(* ADS write *)
_fbWriteProp(
	BACnetDevicePort	:= stAdsConn.nAmsPort,
	bExecute			:= ,
	sNetId				:= stAdsConn.sAmsNetId,
	ObjectType			:= F_BACnet_GetObjType(tObjectID),
	PropertyID			:= BACnetPropertyIdentifier_RecipientList,
	Priority			:= BACnetPriority_None,
	DataType			:= BACnetDataType_RecipientArr,
	ObjectInstance		:= F_BACnet_GetObjInstance(tObjectID),
	ptrValue			:= ADR(stBACnet_AdsBuffer.arrData),
	nLenValue			:= TO_UDINT(_iDataEntry) * TO_UDINT(_cbDestListElem),
	bDone				=> ,
	bBusy				=> ,
	bError				=> ,
	nErrID				=> );

(* trigger start event *)
_rtrigGet(CLK:= bGet, Q=> );
_rtrigSet(CLK:= bSet, Q=> );

(* state machine *)
CASE _i OF

	0: (* Idle *)
		IF 		_rtrigGet.Q
			OR	_rtrigSet.Q
			OR	(		(		(_nAdsReloadOld <> stAdsConn.nReload)
							OR	(_tObjectIDOld <> tObjectID)
						)
					AND	bAutoGet
				)
		THEN
			IF (NOT stAdsConn.bValid) THEN
				(* ADS connection not valid *)
				nErrorId := BACnet_ERR_INVALID_ADS_CONN;
			ELSIF (NOT stAdsConn.bServer AND NOT stAdsConn.bClient) THEN
				(* not a server nor a client *)
				nErrorId := BACnet_ERR_ADS_NoServerClient;
			ELSE
				(* decide get or set *)
				IF _rtrigGet.Q THEN
					_i := 1;
				ELSIF _rtrigSet.Q THEN
					_i := 11;
				ELSIF bAutoGet THEN
					_i := 1;
				END_IF
				nErrorId := BACnet_ERR_NO_ERROR;
				(* reset index *)
				_iEntry	:= 0;
				(* initialize pointer *)
				_pEntryList := ADR(stBACnet_AdsBuffer.arrData);
				(* remind parameter *)
				_tObjectIDOld := tObjectID;
				_nAdsReloadOld := stAdsConn.nReload;
			END_IF
			(* reset done flag *)
			bDone := FALSE;
		END_IF
		IF (NOT bGet) AND (NOT bSet) AND (NOT bAutoGet) THEN
			nErrorId := BACnet_ERR_NO_ERROR;
			bDone := FALSE;
		END_IF

	(* READ *)
	1: (* read object property data via ADS *)
		IF TestAndSet(stBACnet_AdsBuffer.bTestSet) THEN
			IF _fbReadProp.bExecute THEN
				IF _fbReadProp.bError THEN
					_i := 100;
					nErrorId := BACnet_ERR_ADS_Read;
					_fbReadProp.bExecute := FALSE;
				ELSIF (NOT _fbReadProp.bBusy) THEN
					_i := 2;
					_fbReadProp.bExecute := FALSE;
					(* clear output data *)
					MEMSET(ADR(stRecipients), 0, SIZEOF(stRecipients));
					(* check array size *)
					_cbDestList 	:= SIZEOF(_pEntryList^);
					_cbDestListElem	:= SIZEOF(_pEntryList^[0]);
					_iEntryCheck := MIN(_fbReadProp.nProcessedLen, _cbDestList) MOD _cbDestListElem;
					IF (_iEntryCheck <> 0) OR (_cbDestListElem = 0) THEN
						_i := 100;
						nErrorId := BACnet_ERR_ADS_WrongEntrySize;
					ELSE
						(* scan property *)
						_iDataEntry := 0;
						_iReadElems := MIN(32767, MIN(_fbReadProp.nProcessedLen, _cbDestList) / _cbDestListElem);
						FOR _iEntry := 0 TO UDINT_TO_INT(_iReadElems) - 1 DO
							IF		(_pEntryList^[_iEntry].stRecipient.eRecipientChoice = BACnetRecipientChoice_device)
								AND	(F_BACnet_GetObjType(_pEntryList^[_iEntry].stRecipient.tDeviceId) = BACnetObjectType_Device)
							THEN
								stRecipients.arrDestList[_iDataEntry].stFromTime	:= _pEntryList^[_iEntry].stFromTime;
								stRecipients.arrDestList[_iDataEntry].stToTime	:= _pEntryList^[_iEntry].stToTime;
								stRecipients.arrDestList[_iDataEntry].tDeviceId	:= _pEntryList^[_iEntry].stRecipient.tDeviceId;
								stRecipients.arrDestList[_iDataEntry].nProcessId	:= _pEntryList^[_iEntry].nProcessId;
								stRecipients.arrDestList[_iDataEntry].bMonday		:= _F_BACnet_IsBitFieldBitSet(_pEntryList^[_iEntry].nValidDaysFlags, BACnetDaysOfWeekBits_Monday);
								stRecipients.arrDestList[_iDataEntry].bTuesday	:= _F_BACnet_IsBitFieldBitSet(_pEntryList^[_iEntry].nValidDaysFlags, BACnetDaysOfWeekBits_Tuesday);
								stRecipients.arrDestList[_iDataEntry].bWednesday	:= _F_BACnet_IsBitFieldBitSet(_pEntryList^[_iEntry].nValidDaysFlags, BACnetDaysOfWeekBits_Wednesday);
								stRecipients.arrDestList[_iDataEntry].bThursday	:= _F_BACnet_IsBitFieldBitSet(_pEntryList^[_iEntry].nValidDaysFlags, BACnetDaysOfWeekBits_Thursday);
								stRecipients.arrDestList[_iDataEntry].bFriday		:= _F_BACnet_IsBitFieldBitSet(_pEntryList^[_iEntry].nValidDaysFlags, BACnetDaysOfWeekBits_Friday);
								stRecipients.arrDestList[_iDataEntry].bSaturday	:= _F_BACnet_IsBitFieldBitSet(_pEntryList^[_iEntry].nValidDaysFlags, BACnetDaysOfWeekBits_Saturday);
								stRecipients.arrDestList[_iDataEntry].bSunday		:= _F_BACnet_IsBitFieldBitSet(_pEntryList^[_iEntry].nValidDaysFlags, BACnetDaysOfWeekBits_Sunday);
								stRecipients.arrDestList[_iDataEntry].bToNormal	:= _F_BACnet_IsBitFieldBitSet(_pEntryList^[_iEntry].nEventTransBits, BACnetEventTransitionBit_to_normal);
								stRecipients.arrDestList[_iDataEntry].bToOffNormal:= _F_BACnet_IsBitFieldBitSet(_pEntryList^[_iEntry].nEventTransBits, BACnetEventTransitionBit_to_offnormal);
								stRecipients.arrDestList[_iDataEntry].bToFault	:= _F_BACnet_IsBitFieldBitSet(_pEntryList^[_iEntry].nEventTransBits, BACnetEventTransitionBit_to_fault);
								stRecipients.arrDestList[_iDataEntry].bIssueConfirmedNotification	:= _pEntryList^[_iEntry].bIssueConfNot;
								_iDataEntry := _iDataEntry + 1;
							END_IF
						END_FOR
						(* calculate entry count *)
						stRecipients.nEntries := _iDataEntry;
						_i := 100;
					END_IF
				END_IF

			ELSIF (stBACnet_AdsBuffer.iLocked = 0) THEN
				_fbReadProp.bExecute := TRUE;
				(* lock global ADS buffer *)
				stBACnet_AdsBuffer.iLocked := SIZEOF(stBACnet_AdsBuffer.arrData);
			END_IF

			(* release temporary task lock *)
			stBACnet_AdsBuffer.bTestSet := FALSE;
		END_IF


	(* WRITE *)
	11: (* lock global ADS buffer *)
		IF TestAndSet(stBACnet_AdsBuffer.bTestSet) THEN
			IF stBACnet_AdsBuffer.iLocked = 0 THEN
				stBACnet_AdsBuffer.iLocked := SIZEOF(stBACnet_AdsBuffer.arrData);

				(* check array size *)
				_cbDestList 	:= SIZEOF(_pEntryList^);
				_cbDestListElem	:= SIZEOF(_pEntryList^[0]);

				(* scan property *)
				_iDataEntry := 0;
				FOR _iEntry := 0 TO MIN(stRecipients.nEntries - 1, TO_INT(BACnet_MaxDestinationArray)) DO
					IF (F_BACnet_GetObjType(stRecipients.arrDestList[_iEntry].tDeviceId) = BACnetObjectType_Device) THEN
						(* clear buffer *)
						MEMSET(ADR(_pEntryList^[_iDataEntry]), 0, _cbDestListElem);
						(* copy time and recipient information *)
						_pEntryList^[_iDataEntry].stFromTime			:= stRecipients.arrDestList[_iEntry].stFromTime;
						_pEntryList^[_iDataEntry].stToTime				:= stRecipients.arrDestList[_iEntry].stToTime;
						_pEntryList^[_iDataEntry].stRecipient.tDeviceId	:= stRecipients.arrDestList[_iEntry].tDeviceId;
						_pEntryList^[_iDataEntry].nProcessId			:= stRecipients.arrDestList[_iEntry].nProcessId;
						(* set valid days flags *)
						_pEntryList^[_iDataEntry].nValidDaysFlags := DWORD#16#00000001;
						_F_BACnet_ChangeBitFieldBit(ADR(_pEntryList^[_iDataEntry].nValidDaysFlags), BACnetDaysOfWeekBits_Monday, stRecipients.arrDestList[_iEntry].bMonday);
						_F_BACnet_ChangeBitFieldBit(ADR(_pEntryList^[_iDataEntry].nValidDaysFlags), BACnetDaysOfWeekBits_Tuesday, stRecipients.arrDestList[_iEntry].bTuesday);
						_F_BACnet_ChangeBitFieldBit(ADR(_pEntryList^[_iDataEntry].nValidDaysFlags), BACnetDaysOfWeekBits_Wednesday, stRecipients.arrDestList[_iEntry].bWednesday);
						_F_BACnet_ChangeBitFieldBit(ADR(_pEntryList^[_iDataEntry].nValidDaysFlags), BACnetDaysOfWeekBits_Thursday, stRecipients.arrDestList[_iEntry].bThursday);
						_F_BACnet_ChangeBitFieldBit(ADR(_pEntryList^[_iDataEntry].nValidDaysFlags), BACnetDaysOfWeekBits_Friday, stRecipients.arrDestList[_iEntry].bFriday);
						_F_BACnet_ChangeBitFieldBit(ADR(_pEntryList^[_iDataEntry].nValidDaysFlags), BACnetDaysOfWeekBits_Saturday, stRecipients.arrDestList[_iEntry].bSaturday);
						_F_BACnet_ChangeBitFieldBit(ADR(_pEntryList^[_iDataEntry].nValidDaysFlags), BACnetDaysOfWeekBits_Sunday, stRecipients.arrDestList[_iEntry].bSunday);
						(* set event transition flags *)
						_pEntryList^[_iDataEntry].nEventTransBits := DWORD#16#00000005;
						_F_BACnet_ChangeBitFieldBit(ADR(_pEntryList^[_iDataEntry].nEventTransBits), BACnetEventTransitionBit_to_normal, stRecipients.arrDestList[_iEntry].bToNormal);
						_F_BACnet_ChangeBitFieldBit(ADR(_pEntryList^[_iDataEntry].nEventTransBits), BACnetEventTransitionBit_to_offnormal, stRecipients.arrDestList[_iEntry].bToOffNormal);
						_F_BACnet_ChangeBitFieldBit(ADR(_pEntryList^[_iDataEntry].nEventTransBits), BACnetEventTransitionBit_to_fault, stRecipients.arrDestList[_iEntry].bToFault);
						(* set confirmed notification flag *)
						_pEntryList^[_iDataEntry].bIssueConfNot := stRecipients.arrDestList[_iEntry].bIssueConfirmedNotification;
						(* set fix choice recipient choice *)
						_pEntryList^[_iDataEntry].stRecipient.eRecipientChoice := BACnetRecipientChoice_device;
						_iDataEntry := _iDataEntry + 1;
					ELSE
						(* Wrong recipient type (device expected) *)
						nErrorId := BACnet_ERR_ADS_RecipientData;
						_i := 100;
						EXIT;
					END_IF
				END_FOR
				(* send data *)
				_i := 12;
			END_IF
			(* release temporary task lock *)
			stBACnet_AdsBuffer.bTestSet := FALSE;
		END_IF

	12:
		IF _fbWriteProp.bExecute AND (NOT _fbWriteProp.bBusy) THEN
			(* check result *)
			_fbWriteProp.bExecute := FALSE;
			IF _fbWriteProp.bError THEN
				nErrorId := BACnet_ERR_ADS_Write;
			END_IF
			_i := 100;
		ELSE
			(* start ADS write *)
			_fbWriteProp.bExecute := TRUE;
		END_IF

	100: (* Done *)
		bDone := (nErrorId = BACnet_ERR_NO_ERROR);
		(* release ADS buffer *)
		stBACnet_AdsBuffer.iLocked := 0;
		_i := 0;

END_CASE

(* set error flag *)
bError 	:= nErrorId > BACnet_ERR_NO_ERROR;
bBusy 	:= _i > 0;

END_FUNCTION_BLOCK

// POUs/BACnet Helper/[internal]/_F_BACnet_ChangeBitFieldBit
FUNCTION _F_BACnet_ChangeBitFieldBit : DWORD
VAR_INPUT
	ptrData		: POINTER TO DWORD;
	bitNbr			: INT;
	Value		: BOOL;
END_VAR
VAR
END_VAR

IF (NOT Value) THEN
	ptrData^ := ptrData^ AND NOT (SHR(DWORD#16#00008000,_F_BACnet_BitFieldBit(bitNbr)));
ELSE
	ptrData^ := ptrData^ OR (SHR(DWORD#16#00008000,_F_BACnet_BitFieldBit(bitNbr)));
END_IF
_F_BACnet_ChangeBitFieldBit := ptrData^;

END_FUNCTION

// POUs/BACnet ADS/Properties/FB_BACnet_WeeklyScheduleProperty
FUNCTION_BLOCK FB_BACnet_WeeklyScheduleProperty
VAR_INPUT
	tObjectID			: T_BACnet_ObjectIdentifier := 16#FFFFFFFF;
	bAutoGet			: BOOL:=TRUE; (* TRUE = get data from property when ADS connection OR object ID changed *)
	bGet				: BOOL; (* FALSE --> TRUE = get data from property *)
	bSet				: BOOL; (* FALSE --> TRUE = set data into property *)
END_VAR
VAR_IN_OUT
	stWeeklySched		: ST_BACnet_WeeklyScheduleBool;
	stAdsConn			: ST_BACnet_AdsConnection;
END_VAR
VAR_OUTPUT
	bDone				: BOOL;
	bBusy				: BOOL;
	bError				: BOOL;
	nErrorId			: UINT;
END_VAR
VAR
	_fbReadProp		: FB_BACnet_ReadProp;
	_fbWriteProp	: FB_BACnet_WriteProp;
	_i				: INT;
	_pDailySched	: POINTER TO ST_BACnet_DailySchedule;
	_pTimeValue		: POINTER TO ST_BACnet_TimeValueList;
	_pOldTimeValue	: POINTER TO ST_BACnet_TimeValueList;
	_iDayBuffer		: INT;
	_iDayEntryBuf	: INT;
	_rtrigGet		: R_TRIG;
	_rtrigSet		: R_TRIG;

	_cbTmpSize		: UDINT;
	_cbTotalEntry	: UDINT;
	_cbTotalBuf		: UDINT;
	_bNextDay		: BOOL;
	_bNextTimeValue	: BOOL;
	_nDays			: UINT;
	_nAdsReloadOld	: USINT;
	_tObjectIDOld	: T_BACnet_ObjectIdentifier := 16#FFFFFFFF;

END_VAR

(*

Listheader:

typedef struct _ListEntryHdr
{
      DWORD nEntrySize;
      DWORD hdrInfo;
}ListEntryHdr, *PListEntryHdr;

#define ListAlignedSize(n)         (4*(((n)+3)/4))
#define FirstListEntry(p) ( (p)->nEntrySize == 0 )                          ? NULL:p
#define NextListEntry(p) ( ( ((p)->nEntrySize&0x80000000) == 0 ) ? NULL:(PBYTE)(p) + ( ListAlignedSize((p)->nEntrySize&~(0x80000000)) + sizeof(ListEntryHdr)) ) // +4 da für nEntrySize 4 Byte reserviert sind, HighBit ausmaskieren
#define ElemSize(p) ((p)->nEntrySize&(~0x80000000))
#define AlignedEntrySize(p) (ListAlignedSize((p)->nEntrySize&(~0x80000000)))

###################################################################

PropExceptionSchedule:

enum BACnetSpecialEventChoice
{
      calendarEntry,
      calendarReference,
      MaxBACnetSpecialEventChoice
};

typedef struct _BACnetCalendarEntry
{
      BACnetCalendarEntryChoice choice;
      union
      {
            BACnetDate              date;
            BACnetDateRange   dateRange;
            BACnetWeekNDay          weekNDay;
      };
}BACnetCalendarEntry, *PBACnetCalendarEntry;

enum BACnetValueChoice
{
      NullValue                    = 0,
      BoolValue                    = 1,
      UnsignedValue                = 2,
      SignedValue                  = 3,
      RealValue                    = 4,
      DoubleValue                  = 5,
      OctedStringValue        = 6,
      CharStringValue         = 7,
      ObjectIdentifierValue = 8,   // but DataType is 0x0C
      EnumerationValue        = 9,
      MaxBACnetValueChoice    = 10
};

typedef struct _BACnetValue  
{
      BACnetValueChoice choice;
      DWORD                        length;     // Alignment + Datenlänge die folgt
      union
      {
            BOOL                                     boolValue;
            FLOAT                                    realValue;
            DOUBLE                                   doubleValue;
            INT                                      signedValue;
            UINT                                     unsignedValue;
            BYTE*                                    pOctedStringValue; 
            CHAR*                                    pCharStringValue;
            BACnetObjectIdentifier  objectIdentifierValue;
            EnumerationValueType         enumerationValue;
      };
}BACnetValue, *PBACnetValue;

typedef struct _BACnetTimeValue
{
      BACnetTime time;
      DWORD  reserved;  // 64bit Alignment
      BACnetValue value;
}BACnetTimeValue, *PBACnetTimeValue;

typedef struct _BACnetTimeValueList
{
      DWORD nEntrySize; // 0x80000000 -> next entry
      DWORD reserved;
      BACnetTimeValue listEntry;
}BACnetTimeValueList, *PBACnetTimeValueList;

typedef struct _BACnetSpecialEvent
{
      BACnetSpecialEventChoice choice;
      union
      {
            BACnetCalendarEntry calendarEntry;
            BACnetObjectIdentifier calendarReference;
      };
      DWORD eventPriority; // DWORD due to alignment
      DWORD reserved;
      BACnetTimeValueList listOfTimeValues;
}BACnetSpecialEvent, *PBACnetSpecialEvent;

typedef struct _BACnetSpecialEventList
{
      DWORD nEntrySize; // 0x80000000 -> next entry
      DWORD reserved;
      BACnetSpecialEvent listEntry;
}BACnetSpecialEventList, *PBACnetSpecialEventList;

###################################################################

PropWeeklySchedule:

typedef struct _BACnetDailySchedule
{
      DWORD nEntrySize; // 0x80000000 -> next entry
      DWORD reserved;
      BACnetTimeValueList listEntry;
} BACnetDailySchedule, *PBACnetDailySchedule;

###################################################################

PropScheduleDefault / PropPresentValue

typedef struct _BACnetValueList
{
      DWORD nEntrySize; // 0x80000000 -> next entry
      DWORD reserved;
      BACnetValue listEntry;
} BACnetValueList, *PBACnetValueList;

###################################################################

*)

(* ADS read *)
_fbReadProp(
	BACnetDevicePort	:= stAdsConn.nAmsPort,
	bExecute			:= ,
	sNetId				:= stAdsConn.sAmsNetId,
	ObjectType			:= F_BACnet_GetObjType(tObjectID),
	PropertyID			:= BACnetPropertyIdentifier_WeeklySchedule,
	DataType			:= BACnetDataType_DailyScheduleList,
	ObjectInstance		:= F_BACnet_GetObjInstance(tObjectID),
	ptrValue			:= ADR(stBACnet_AdsBuffer.arrData),
	nLenValue			:= SIZEOF(stBACnet_AdsBuffer.arrData),
	bDone				=> ,
	bBusy				=> ,
	bError				=> ,
	nErrID				=> ,
	nProcessedLen		=> );

_fbWriteProp(
	BACnetDevicePort	:= stAdsConn.nAmsPort,
	bExecute			:= ,
	sNetId				:= stAdsConn.sAmsNetId,
	ObjectType			:= F_BACnet_GetObjType(tObjectID),
	PropertyID			:= BACnetPropertyIdentifier_WeeklySchedule,
	Priority			:= BACnetPriority_None,
	DataType			:= BACnetDataType_DailyScheduleList,
	ObjectInstance		:= F_BACnet_GetObjInstance(tObjectID),
	ptrValue			:= ADR(stBACnet_AdsBuffer.arrData),
	nLenValue			:= _cbTotalBuf,
	bDone				=> ,
	bBusy				=> ,
	bError				=> ,
	nErrID				=> );

(* trigger start event *)
_rtrigGet(CLK:= bGet, Q=> );
_rtrigSet(CLK:= bSet, Q=> );

(* state machine *)
CASE _i OF

	0: (* Idle *)
		IF 		_rtrigGet.Q
			OR	_rtrigSet.Q
			OR	(		(		(_nAdsReloadOld <> stAdsConn.nReload)
							OR	(_tObjectIDOld <> tObjectID)
						)
					AND	bAutoGet
				)
			OR	stWeeklySched.bReqGet
			OR	stWeeklySched.bReqSet
		THEN
			IF (NOT stAdsConn.bValid) THEN
				(* ADS connection not valid *)
				nErrorId := BACnet_ERR_INVALID_ADS_CONN;
			ELSIF (NOT stAdsConn.bServer AND NOT stAdsConn.bClient) THEN
				(* not a server nor a client *)
				nErrorId := BACnet_ERR_ADS_NoServerClient;
			ELSE
				(* check day count *)
				_nDays := SIZEOF(stWeeklySched.arrEntries) / SIZEOF(stWeeklySched.arrEntries[0]);
				(* decide get or set *)
				IF _rtrigGet.Q OR stWeeklySched.bReqGet THEN
					_i := 1;
					stWeeklySched.bReqGet := FALSE;
				ELSIF _rtrigSet.Q OR stWeeklySched.bReqSet THEN
					_i := 11;
					stWeeklySched.bReqSet := FALSE;
				ELSIF bAutoGet THEN
					_i := 1;
					stWeeklySched.bReqGet := FALSE;
				END_IF
				nErrorId := BACnet_ERR_NO_ERROR;
				(* remind parameter *)
				_tObjectIDOld := tObjectID;
				_nAdsReloadOld := stAdsConn.nReload;
				(* lock data array *)
				stWeeklySched.bBusy := TRUE;
			END_IF
			(* reset done flag *)
			bDone := FALSE;
		END_IF
		IF (NOT bGet) AND (NOT bSet) AND (NOT bAutoGet) THEN
			nErrorId := BACnet_ERR_NO_ERROR;
			bDone := FALSE;
		END_IF

	(* READ *)
	1: (* read object property data over ADS *)
		IF TestAndSet(stBACnet_AdsBuffer.bTestSet) THEN
			IF _fbReadProp.bExecute THEN
				IF _fbReadProp.bError THEN
					_i := 100;
					nErrorId := BACnet_ERR_ADS_Read;
					_fbReadProp.bExecute := FALSE;
				ELSIF (NOT _fbReadProp.bBusy) THEN
					_i := 2;
					_fbReadProp.bExecute := FALSE;
					_pDailySched := ADR(stBACnet_AdsBuffer.arrData);
					MEMSET(ADR(stWeeklySched.arrEntries), 0, SIZEOF(stWeeklySched.arrEntries));
					_iDayBuffer := 0;
					_cbTotalBuf := 0;
				END_IF
			ELSE
				(* lock global ADS buffer and start reading *)
				IF stBACnet_AdsBuffer.iLocked = 0 THEN
					_fbReadProp.bExecute := TRUE;
					stBACnet_AdsBuffer.iLocked := SIZEOF(stBACnet_AdsBuffer.arrData);
				END_IF
			END_IF

			(* release temporary task lock *)
			stBACnet_AdsBuffer.bTestSet := FALSE;
		END_IF

	2: (* select day *)
		_pTimeValue := ADR(_pDailySched^.stListEntry);
		(* scan time value list *)
		_iDayEntryBuf := 0;
		_i := 3;

	3: (* select time value *)
		WHILE (_i = 3) DO
			(* check entry size of time value *)
			IF (_pTimeValue^.nEntrySize AND 16#7FFFFFFF) > 0 THEN
				(* check internal schedule buffer index *)
				IF (_iDayBuffer > TO_INT(_nDays)-1) THEN
					(* error, wrong day index *)
					nErrorId := BACnet_ERR_ADS_SchedData;
					_i := 100;
				ELSE
					IF (_iDayEntryBuf <= TO_INT(BACnet_MaxDayEntry)) THEN
						IF _pTimeValue^.stListEntry.stValue.eValueChoice = BACnetDataType_Null THEN
							(* NULL *)
							stWeeklySched.arrEntries[_iDayBuffer][_iDayEntryBuf].stTime	:= _pTimeValue^.stListEntry.stTime;
							stWeeklySched.arrEntries[_iDayBuffer][_iDayEntryBuf].eType		:= _pTimeValue^.stListEntry.stValue.eValueChoice;
							stWeeklySched.arrEntries[_iDayBuffer][_iDayEntryBuf].bValue	:= FALSE;
							stWeeklySched.arrEntries[_iDayBuffer][_iDayEntryBuf].bValid	:= TRUE;
							_iDayEntryBuf := _iDayEntryBuf + 1;

						ELSIF (_pTimeValue^.stListEntry.stValue.cbData = 1) THEN
							(* read time, data type and value *)
							stWeeklySched.arrEntries[_iDayBuffer][_iDayEntryBuf].stTime	:= _pTimeValue^.stListEntry.stTime;
							stWeeklySched.arrEntries[_iDayBuffer][_iDayEntryBuf].eType		:= _pTimeValue^.stListEntry.stValue.eValueChoice;
							stWeeklySched.arrEntries[_iDayBuffer][_iDayEntryBuf].bValue	:= FALSE;
							MEMCPY(	ADR(stWeeklySched.arrEntries[_iDayBuffer][_iDayEntryBuf].bValue),
									ADR(_pTimeValue^.stListEntry.stValue.nData),
									MIN(	SIZEOF(stWeeklySched.arrEntries[_iDayBuffer][_iDayEntryBuf].bValue),
											_pTimeValue^.stListEntry.stValue.cbData
										)
							);
							stWeeklySched.arrEntries[_iDayBuffer][_iDayEntryBuf].bValid	:= TRUE;
							_iDayEntryBuf := _iDayEntryBuf + 1;
						ELSE
							(* unsupported data type length *);
						END_IF
					END_IF

					(* next time value entry *)
					_NextTimeValue();
					(* check if next time value entry available *)
					IF (NOT _bNextTimeValue) THEN
						(* update pointer each cycle (even if no day follows!) *)
						_NextDay();
						(* check for next day *)
						IF _bNextDay THEN
							(* go on *)
							_iDayBuffer := _iDayBuffer + 1;
							_i := 2;
						ELSE
							(* DONE *)
							_i := 4;
						END_IF
					END_IF
				END_IF

			ELSE
				(* update pointer each cycle (even if no day follows!) *)
				_NextDay();
				(* No timevalue entry, check if next day element exists and pointer is plausible *)
				IF _bNextDay THEN
					(* next day entry exists, go on *)
					_iDayBuffer := _iDayBuffer + 1;
					(* check pointer *)
					IF (_pDailySched + (_pDailySched^.nEntrySize AND 16#7FFFFFFF)) < (ADR(stBACnet_AdsBuffer.arrData) + SIZEOF(stBACnet_AdsBuffer.arrData)) THEN
						_i := 2;
					ELSE
						(* buffer too small *)
						nErrorId := BACnet_ERR_ADS_BufferSize;
						_i := 100;
					END_IF
				ELSE
					(* DONE *)
					_i := 4;
				END_IF
			END_IF
		END_WHILE

	4: (* data read and parsed successful *)
		stWeeklySched.nGet := stWeeklySched.nGet +1;
		_i := 100;

	(* WRITE *)
	11: (* lock global ADS buffer *)
		IF TestAndSet(stBACnet_AdsBuffer.bTestSet) THEN
			IF stBACnet_AdsBuffer.iLocked = 0 THEN
				stBACnet_AdsBuffer.iLocked := SIZEOF(stBACnet_AdsBuffer.arrData);
				_i := 12;
				(*MEMSET(ADR(stBACnet_AdsBuffer.arrData), 0, SIZEOF(stBACnet_AdsBuffer.arrData));*)
			END_IF
			(* release temporary task lock *)
			stBACnet_AdsBuffer.bTestSet := FALSE;
		END_IF

	12: (* prepare data *)
		(* set day pointer *)
		_pDailySched := ADR(stBACnet_AdsBuffer.arrData);
		_cbTotalBuf := 0;
		(* scan schedule data *)
		FOR _iDayBuffer := 0 TO TO_INT(_nDays)-1 DO
			(* set timevalue pointer *)
			_pTimeValue := ADR(_pDailySched^.stListEntry);
			_cbTotalEntry := 0;
			_pOldTimeValue := 0;
			(* scan time values *)
			FOR _iDayEntryBuf := 0 TO TO_INT(BACnet_MaxDayEntry) DO
				IF		stWeeklySched.arrEntries[_iDayBuffer][_iDayEntryBuf].bValid
					AND	(		stWeeklySched.arrEntries[_iDayBuffer][_iDayEntryBuf].eType = BACnetDataType_Bool
							OR	stWeeklySched.arrEntries[_iDayBuffer][_iDayEntryBuf].eType = BACnetDataType_Null
						)
				THEN
					(* set flag "next entry" to the previous element *)
					IF (_iDayEntryBuf > 0) AND (_pOldTimeValue <> 0) THEN
						_pOldTimeValue^.nEntrySize := _pOldTimeValue^.nEntrySize + 16#80000000;
					END_IF
					(* set data *)
					_pTimeValue^.stListEntry.stValue.nData := 0; (* clear data *)
					_pTimeValue^.stListEntry.stTime := stWeeklySched.arrEntries[_iDayBuffer][_iDayEntryBuf].stTime;
					(* decide between None and Bool type *)
					IF stWeeklySched.arrEntries[_iDayBuffer][_iDayEntryBuf].eType = BACnetDataType_Bool THEN
						_pTimeValue^.stListEntry.stValue.cbData := SIZEOF(stWeeklySched.arrEntries[_iDayBuffer][_iDayEntryBuf].bValue);
						_pTimeValue^.stListEntry.stValue.eValueChoice := BACnetDataType_Bool;
						_pTimeValue^.stListEntry.stValue.nRes1 := 0;
						MEMCPY(	ADR(_pTimeValue^.stListEntry.stValue.nData),
								ADR(stWeeklySched.arrEntries[_iDayBuffer][_iDayEntryBuf].bValue),
								1
						);
					ELSE
						(* unsupported *)
						_pTimeValue^.stListEntry.stValue.cbData := 0;
						_pTimeValue^.stListEntry.stValue.eValueChoice := BACnetDataType_Null;
						_pTimeValue^.stListEntry.stValue.nRes1 := 0;
					END_IF

					(* calculate time-value entry size *)
					_pTimeValue^.nEntrySize :=	_pTimeValue^.stListEntry.stValue.cbData
											+	SIZEOF(_pTimeValue^.stListEntry.nRes)
											+	SIZEOF(_pTimeValue^.stListEntry.stTime)
											+	SIZEOF(_pTimeValue^.stListEntry.stValue.cbData)
											+	SIZEOF(_pTimeValue^.stListEntry.stValue.eValueChoice)
											+	SIZEOF(_pTimeValue^.stListEntry.stValue.nRes1);

					(* update time value pointer *)
					_NextTimeValue();

					(* ...and add to total entry size counter *)
					_cbTotalEntry := _cbTotalEntry + _cbTmpSize;
				ELSE
					(* reset time value entry *)
					_pTimeValue^.nEntrySize := 0;
					_pTimeValue^.stListEntry.stValue.cbData := 0;
					_pTimeValue^.stListEntry.stValue.nRes1 := 0;
				END_IF
			END_FOR

			(* caclulate day-entry size *)
			_pDailySched^.nEntrySize := MAX(_cbTotalEntry, SIZEOF(_pDailySched^.stListEntry.nEntrySize) + SIZEOF(_pDailySched^.stListEntry.nRes));

			(* next day? *)
			IF (_iDayBuffer < to_int(_nDays)-1) THEN
				_pDailySched^.nEntrySize := _pDailySched^.nEntrySize + 16#80000000;
			END_IF

			(* update pointer each cycle (even if no day follows!) *)
			_NextDay();
		END_FOR
		(* send data *)
		_i := 13;

	13:
		IF _fbWriteProp.bExecute AND (NOT _fbWriteProp.bBusy) THEN
			(* check result *)
			_fbWriteProp.bExecute := FALSE;
			IF _fbWriteProp.bError THEN
				nErrorId := BACnet_ERR_ADS_Write;
			ELSE
				stWeeklySched.nSet := stWeeklySched.nSet +1;
			END_IF
			_i := 100;
		ELSE
			(* start ADS write *)
			_fbWriteProp.bExecute := TRUE;
		END_IF

	100: (* Done *)
		bDone := (nErrorId = BACnet_ERR_NO_ERROR);
		(* release ADS buffer *)
		stBACnet_AdsBuffer.iLocked := 0;
		(* release data array *)
		stWeeklySched.bBusy := FALSE;
		(* go idle *)
		_i := 0;

END_CASE

(* set error flag *)
bError 	:= nErrorId > BACnet_ERR_NO_ERROR;
bBusy 	:= _i > 0;

ACTION _NextDay:
_bNextDay := ((_pDailySched^.nEntrySize AND 16#80000000) = 16#80000000);
_cbTmpSize := _F_BACnet_AlignedSize(_pDailySched^.nEntrySize AND 16#7FFFFFFF) + SIZEOF(_pDailySched^.nEntrySize) + SIZEOF(_pDailySched^.nRes);
_pDailySched := _pDailySched + _cbTmpSize;
_cbTotalBuf := _cbTotalBuf + _cbTmpSize;
_pOldTimeValue := 0;
END_ACTION

ACTION _NextTimeValue:
_bNextTimeValue := (_pTimeValue^.nEntrySize AND 16#80000000) = 16#80000000;
_cbTmpSize := _F_BACnet_AlignedSize(_pTimeValue^.nEntrySize AND 16#7FFFFFFF) + SIZEOF(_pDailySched^.stListEntry.nEntrySize) + SIZEOF(_pDailySched^.stListEntry.nRes);
_pOldTimeValue := _pTimeValue;
_pTimeValue := _pTimeValue + _cbTmpSize;
END_ACTION

END_FUNCTION_BLOCK

// POUs/BACnet ADS/Properties/FB_BACnet_WeeklySchedulePropertyReal
FUNCTION_BLOCK FB_BACnet_WeeklySchedulePropertyReal
VAR_INPUT
	tObjectID			: T_BACnet_ObjectIdentifier := 16#FFFFFFFF;
	bAutoGet			: BOOL:=TRUE; (* TRUE = get data from property when ADS connection OR object ID changed *)
	bGet				: BOOL; (* FALSE --> TRUE = get data from property *)
	bSet				: BOOL; (* FALSE --> TRUE = set data into property *)
END_VAR
VAR_IN_OUT
	stWeeklySched		: ST_BACnet_WeeklyScheduleReal;
	stAdsConn			: ST_BACnet_AdsConnection;
END_VAR
VAR_OUTPUT
	bDone				: BOOL;
	bBusy				: BOOL;
	bError				: BOOL;
	nErrorId			: UINT;
END_VAR
VAR
	_fbReadProp		: FB_BACnet_ReadProp;
	_fbWriteProp	: FB_BACnet_WriteProp;
	_i				: INT;
	_pDailySched	: POINTER TO ST_BACnet_DailySchedule;
	_pTimeValue		: POINTER TO ST_BACnet_TimeValueList;
	_pOldTimeValue	: POINTER TO ST_BACnet_TimeValueList;
	_iDayBuffer		: INT;
	_iDayEntryBuf	: INT;
	_rtrigGet		: R_TRIG;
	_rtrigSet		: R_TRIG;

	_cbTmpSize		: UDINT;
	_cbTotalEntry	: UDINT;
	_cbTotalBuf		: UDINT;
	_bNextDay		: BOOL;
	_bNextTimeValue	: BOOL;
	_nDays			: UINT;
	_nAdsReloadOld	: USINT;
	_tObjectIDOld	: T_BACnet_ObjectIdentifier := 16#FFFFFFFF;

	_pReal			: POINTER TO REAL;
END_VAR

(*

Listheader:

typedef struct _ListEntryHdr
{
      DWORD nEntrySize;
      DWORD hdrInfo;
}ListEntryHdr, *PListEntryHdr;

#define ListAlignedSize(n)         (4*(((n)+3)/4))
#define FirstListEntry(p) ( (p)->nEntrySize == 0 )                          ? NULL:p
#define NextListEntry(p) ( ( ((p)->nEntrySize&0x80000000) == 0 ) ? NULL:(PBYTE)(p) + ( ListAlignedSize((p)->nEntrySize&~(0x80000000)) + sizeof(ListEntryHdr)) ) // +4 da für nEntrySize 4 Byte reserviert sind, HighBit ausmaskieren
#define ElemSize(p) ((p)->nEntrySize&(~0x80000000))
#define AlignedEntrySize(p) (ListAlignedSize((p)->nEntrySize&(~0x80000000)))

###################################################################

PropExceptionSchedule:

enum BACnetSpecialEventChoice
{
      calendarEntry,
      calendarReference,
      MaxBACnetSpecialEventChoice
};

typedef struct _BACnetCalendarEntry
{
      BACnetCalendarEntryChoice choice;
      union
      {
            BACnetDate              date;
            BACnetDateRange   dateRange;
            BACnetWeekNDay          weekNDay;
      };
}BACnetCalendarEntry, *PBACnetCalendarEntry;

enum BACnetValueChoice
{
      NullValue                    = 0,
      BoolValue                    = 1,
      UnsignedValue                = 2,
      SignedValue                  = 3,
      RealValue                    = 4,
      DoubleValue                  = 5,
      OctedStringValue        = 6,
      CharStringValue         = 7,
      ObjectIdentifierValue = 8,   // but DataType is 0x0C
      EnumerationValue        = 9,
      MaxBACnetValueChoice    = 10
};

typedef struct _BACnetValue  
{
      BACnetValueChoice choice;
      DWORD                        length;     // Alignment + Datenlänge die folgt
      union
      {
            BOOL                                     boolValue;
            FLOAT                                    realValue;
            DOUBLE                                   doubleValue;
            INT                                      signedValue;
            UINT                                     unsignedValue;
            BYTE*                                    pOctedStringValue; 
            CHAR*                                    pCharStringValue;
            BACnetObjectIdentifier  objectIdentifierValue;
            EnumerationValueType         enumerationValue;
      };
}BACnetValue, *PBACnetValue;

typedef struct _BACnetTimeValue
{
      BACnetTime time;
      DWORD  reserved;  // 64bit Alignment
      BACnetValue value;
}BACnetTimeValue, *PBACnetTimeValue;

typedef struct _BACnetTimeValueList
{
      DWORD nEntrySize; // 0x80000000 -> next entry
      DWORD reserved;
      BACnetTimeValue listEntry;
}BACnetTimeValueList, *PBACnetTimeValueList;

typedef struct _BACnetSpecialEvent
{
      BACnetSpecialEventChoice choice;
      union
      {
            BACnetCalendarEntry calendarEntry;
            BACnetObjectIdentifier calendarReference;
      };
      DWORD eventPriority; // DWORD due to alignment
      DWORD reserved;
      BACnetTimeValueList listOfTimeValues;
}BACnetSpecialEvent, *PBACnetSpecialEvent;

typedef struct _BACnetSpecialEventList
{
      DWORD nEntrySize; // 0x80000000 -> next entry
      DWORD reserved;
      BACnetSpecialEvent listEntry;
}BACnetSpecialEventList, *PBACnetSpecialEventList;

###################################################################

PropWeeklySchedule:

typedef struct _BACnetDailySchedule
{
      DWORD nEntrySize; // 0x80000000 -> next entry
      DWORD reserved;
      BACnetTimeValueList listEntry;
} BACnetDailySchedule, *PBACnetDailySchedule;

###################################################################

PropScheduleDefault / PropPresentValue

typedef struct _BACnetValueList
{
      DWORD nEntrySize; // 0x80000000 -> next entry
      DWORD reserved;
      BACnetValue listEntry;
} BACnetValueList, *PBACnetValueList;

###################################################################

*)

(* ADS read *)
_fbReadProp(
	BACnetDevicePort	:= stAdsConn.nAmsPort,
	bExecute			:= ,
	sNetId				:= stAdsConn.sAmsNetId,
	ObjectType			:= F_BACnet_GetObjType(tObjectID),
	PropertyID			:= BACnetPropertyIdentifier_WeeklySchedule,
	DataType			:= BACnetDataType_DailyScheduleList,
	ObjectInstance		:= F_BACnet_GetObjInstance(tObjectID),
	ptrValue			:= ADR(stBACnet_AdsBuffer.arrData),
	nLenValue			:= SIZEOF(stBACnet_AdsBuffer.arrData),
	bDone				=> ,
	bBusy				=> ,
	bError				=> ,
	nErrID				=> ,
	nProcessedLen		=> );

_fbWriteProp(
	BACnetDevicePort	:= stAdsConn.nAmsPort,
	bExecute			:= ,
	sNetId				:= stAdsConn.sAmsNetId,
	ObjectType			:= F_BACnet_GetObjType(tObjectID),
	PropertyID			:= BACnetPropertyIdentifier_WeeklySchedule,
	Priority			:= BACnetPriority_None,
	DataType			:= BACnetDataType_DailyScheduleList,
	ObjectInstance		:= F_BACnet_GetObjInstance(tObjectID),
	ptrValue			:= ADR(stBACnet_AdsBuffer.arrData),
	nLenValue			:= _cbTotalBuf,
	bDone				=> ,
	bBusy				=> ,
	bError				=> ,
	nErrID				=> );

(* trigger start event *)
_rtrigGet(CLK:= bGet, Q=> );
_rtrigSet(CLK:= bSet, Q=> );

(* state machine *)
CASE _i OF

	0: (* Idle *)
		IF 		_rtrigGet.Q
			OR	_rtrigSet.Q
			OR	(		(		(_nAdsReloadOld <> stAdsConn.nReload)
							OR	(_tObjectIDOld <> tObjectID)
						)
					AND	bAutoGet
				)
			OR	stWeeklySched.bReqGet
			OR	stWeeklySched.bReqSet
		THEN
			IF (NOT stAdsConn.bValid) THEN
				(* ADS connection not valid *)
				nErrorId := BACnet_ERR_INVALID_ADS_CONN;
			ELSIF (NOT stAdsConn.bServer AND NOT stAdsConn.bClient) THEN
				(* not a server nor a client *)
				nErrorId := BACnet_ERR_ADS_NoServerClient;
			ELSE
				(* check day count *)
				_nDays := SIZEOF(stWeeklySched.arrEntries) / SIZEOF(stWeeklySched.arrEntries[0]);
				(* decide get or set *)
				IF _rtrigGet.Q OR stWeeklySched.bReqGet THEN
					_i := 1;
					stWeeklySched.bReqGet := FALSE;
				ELSIF _rtrigSet.Q OR stWeeklySched.bReqSet THEN
					_i := 11;
					stWeeklySched.bReqSet := FALSE;
				ELSIF bAutoGet THEN
					_i := 1;
					stWeeklySched.bReqGet := FALSE;
				END_IF
				nErrorId := BACnet_ERR_NO_ERROR;
				(* remind parameter *)
				_tObjectIDOld := tObjectID;
				_nAdsReloadOld := stAdsConn.nReload;
				(* lock data array *)
				stWeeklySched.bBusy := TRUE;
			END_IF
			(* reset done flag *)
			bDone := FALSE;
		END_IF
		IF (NOT bGet) AND (NOT bSet) AND (NOT bAutoGet) THEN
			nErrorId := BACnet_ERR_NO_ERROR;
			bDone := FALSE;
		END_IF

	(* READ *)
	1: (* read object property data over ADS *)
		IF TestAndSet(stBACnet_AdsBuffer.bTestSet) THEN
			IF _fbReadProp.bExecute THEN
				IF _fbReadProp.bError THEN
					_i := 100;
					nErrorId := BACnet_ERR_ADS_Read;
					_fbReadProp.bExecute := FALSE;
				ELSIF (NOT _fbReadProp.bBusy) THEN
					_i := 2;
					_fbReadProp.bExecute := FALSE;
					_pDailySched := ADR(stBACnet_AdsBuffer.arrData);
					MEMSET(ADR(stWeeklySched.arrEntries), 0, SIZEOF(stWeeklySched.arrEntries));
					_iDayBuffer := 0;
					_cbTotalBuf := 0;
				END_IF
			ELSE
				(* lock global ADS buffer and start reading *)
				IF stBACnet_AdsBuffer.iLocked = 0 THEN
					_fbReadProp.bExecute := TRUE;
					stBACnet_AdsBuffer.iLocked := SIZEOF(stBACnet_AdsBuffer.arrData);
				END_IF
			END_IF

			(* release temporary task lock *)
			stBACnet_AdsBuffer.bTestSet := FALSE;
		END_IF

	2: (* select day *)
		_pTimeValue := ADR(_pDailySched^.stListEntry);
		(* scan time value list *)
		_iDayEntryBuf := 0;
		_i := 3;

	3: (* select time value *)
		WHILE (_i = 3) DO
			(* check entry size of time value *)
			IF (_pTimeValue^.nEntrySize AND 16#7FFFFFFF) > 0 THEN
				(* check internal schedule buffer index *)
				IF (_iDayBuffer > TO_INT(_nDays)-1) THEN
					(* error, wrong day index *)
					nErrorId := BACnet_ERR_ADS_SchedData;
					_i := 100;
				ELSE
					IF (_iDayEntryBuf <= TO_INT(BACnet_MaxDayEntry)) THEN
						IF _pTimeValue^.stListEntry.stValue.eValueChoice = BACnetDataType_Null THEN
							(* NULL *)
							stWeeklySched.arrEntries[_iDayBuffer][_iDayEntryBuf].stTime	:= _pTimeValue^.stListEntry.stTime;
							stWeeklySched.arrEntries[_iDayBuffer][_iDayEntryBuf].eType		:= _pTimeValue^.stListEntry.stValue.eValueChoice;
							stWeeklySched.arrEntries[_iDayBuffer][_iDayEntryBuf].rValue	:= F_BACnet_NAN();
							stWeeklySched.arrEntries[_iDayBuffer][_iDayEntryBuf].bValid	:= TRUE;
							_iDayEntryBuf := _iDayEntryBuf + 1;

						ELSIF (_pTimeValue^.stListEntry.stValue.cbData = 4) THEN
							(* read time, data type and value *)
							stWeeklySched.arrEntries[_iDayBuffer][_iDayEntryBuf].stTime	:= _pTimeValue^.stListEntry.stTime;
							stWeeklySched.arrEntries[_iDayBuffer][_iDayEntryBuf].eType		:= _pTimeValue^.stListEntry.stValue.eValueChoice;
							stWeeklySched.arrEntries[_iDayBuffer][_iDayEntryBuf].rValue	:= F_BACnet_NAN();
							MEMCPY(	ADR(stWeeklySched.arrEntries[_iDayBuffer][_iDayEntryBuf].rValue),
									ADR(_pTimeValue^.stListEntry.stValue.nData),
									MIN(	SIZEOF(stWeeklySched.arrEntries[_iDayBuffer][_iDayEntryBuf].rValue),
											_pTimeValue^.stListEntry.stValue.cbData
										)
							);
							stWeeklySched.arrEntries[_iDayBuffer][_iDayEntryBuf].bValid	:= TRUE;
							_iDayEntryBuf := _iDayEntryBuf + 1;
						ELSE
							(* unsupported data type length *);
						END_IF
					END_IF

					(* next time value entry *)
					_NextTimeValue();
					(* check if next time value entry available *)
					IF (NOT _bNextTimeValue) THEN
						(* update pointer each cycle (even if no day follows!) *)
						_NextDay();
						(* check for next day *)
						IF _bNextDay THEN
							(* go on *)
							_iDayBuffer := _iDayBuffer + 1;
							_i := 2;
						ELSE
							(* DONE *)
							_i := 4;
						END_IF
					END_IF
				END_IF

			ELSE
				(* update pointer each cycle (even if no day follows!) *)
				_NextDay();
				(* No timevalue entry, check if next day element exists and pointer is plausible *)
				IF _bNextDay THEN
					(* next day entry exists, go on *)
					_iDayBuffer := _iDayBuffer + 1;
					(* check pointer *)
					IF (_pDailySched + (_pDailySched^.nEntrySize AND 16#7FFFFFFF)) < (ADR(stBACnet_AdsBuffer.arrData) + SIZEOF(stBACnet_AdsBuffer.arrData)) THEN
						_i := 2;
					ELSE
						(* buffer too small *)
						nErrorId := BACnet_ERR_ADS_BufferSize;
						_i := 100;
					END_IF
				ELSE
					(* DONE *)
					_i := 4;
				END_IF
			END_IF
		END_WHILE

	4: (* data read and parsed successful *)
		stWeeklySched.nGet := stWeeklySched.nGet +1;
		_i := 100;

	(* WRITE *)
	11: (* lock global ADS buffer *)
		IF TestAndSet(stBACnet_AdsBuffer.bTestSet) THEN
			IF stBACnet_AdsBuffer.iLocked = 0 THEN
				stBACnet_AdsBuffer.iLocked := SIZEOF(stBACnet_AdsBuffer.arrData);
				_i := 12;
				(*MEMSET(ADR(stBACnet_AdsBuffer.arrData), 0, SIZEOF(stBACnet_AdsBuffer.arrData));*)
			END_IF
			(* release temporary task lock *)
			stBACnet_AdsBuffer.bTestSet := FALSE;
		END_IF

	12: (* prepare data *)
		(* set day pointer *)
		_pDailySched := ADR(stBACnet_AdsBuffer.arrData);
		_cbTotalBuf := 0;
		(* scan schedule data *)
		FOR _iDayBuffer := 0 TO TO_INT(_nDays)-1 DO
			(* set timevalue pointer *)
			_pTimeValue := ADR(_pDailySched^.stListEntry);
			_cbTotalEntry := 0;
			_pOldTimeValue := 0;
			(* scan time values *)
			FOR _iDayEntryBuf := 0 TO TO_INT(BACnet_MaxDayEntry) DO
				IF		stWeeklySched.arrEntries[_iDayBuffer][_iDayEntryBuf].bValid
					AND	(		stWeeklySched.arrEntries[_iDayBuffer][_iDayEntryBuf].eType = BACnetDataType_Real
							OR	stWeeklySched.arrEntries[_iDayBuffer][_iDayEntryBuf].eType = BACnetDataType_Null
						)
				THEN
					(* set flag "next entry" to the previous element *)
					IF (_iDayEntryBuf > 0) AND (_pOldTimeValue <> 0) THEN
						_pOldTimeValue^.nEntrySize := _pOldTimeValue^.nEntrySize + 16#80000000;
					END_IF
					(* set data *)
					_pReal := ADR(_pTimeValue^.stListEntry.stValue.nData);
					_pReal^ := 0.0; (* clear data *)
					_pTimeValue^.stListEntry.stTime := stWeeklySched.arrEntries[_iDayBuffer][_iDayEntryBuf].stTime;
					(* decide between None and Real type *)
					IF stWeeklySched.arrEntries[_iDayBuffer][_iDayEntryBuf].eType = BACnetDataType_Real THEN
						_pTimeValue^.stListEntry.stValue.cbData := SIZEOF(stWeeklySched.arrEntries[_iDayBuffer][_iDayEntryBuf].rValue);
						_pTimeValue^.stListEntry.stValue.eValueChoice := BACnetDataType_Real;
						_pTimeValue^.stListEntry.stValue.nRes1 := 0;
						MEMCPY(	_pReal,
								ADR(stWeeklySched.arrEntries[_iDayBuffer][_iDayEntryBuf].rValue),
								4
						);
					ELSE
						(* unsupported *)
						_pTimeValue^.stListEntry.stValue.cbData := 0;
						_pTimeValue^.stListEntry.stValue.eValueChoice := BACnetDataType_Null;
						_pTimeValue^.stListEntry.stValue.nRes1 := 0;
					END_IF

					(* calculate time-value entry size *)
					_pTimeValue^.nEntrySize :=	_pTimeValue^.stListEntry.stValue.cbData
											+	SIZEOF(_pTimeValue^.stListEntry.nRes)
											+	SIZEOF(_pTimeValue^.stListEntry.stTime)
											+	SIZEOF(_pTimeValue^.stListEntry.stValue.cbData)
											+	SIZEOF(_pTimeValue^.stListEntry.stValue.eValueChoice)
											+	SIZEOF(_pTimeValue^.stListEntry.stValue.nRes1);

					(* update time value pointer *)
					_NextTimeValue();

					(* ...and add to total entry size counter *)
					_cbTotalEntry := _cbTotalEntry + _cbTmpSize;
				ELSE
					(* reset time value entry *)
					_pTimeValue^.nEntrySize := 0;
					_pTimeValue^.stListEntry.stValue.cbData := 0;
					_pTimeValue^.stListEntry.stValue.nRes1 := 0;
				END_IF
			END_FOR

			(* caclulate day-entry size *)
			_pDailySched^.nEntrySize := MAX(_cbTotalEntry, SIZEOF(_pDailySched^.stListEntry.nEntrySize) + SIZEOF(_pDailySched^.stListEntry.nRes));

			(* next day? *)
			IF (_iDayBuffer < to_int(_nDays)-1) THEN
				_pDailySched^.nEntrySize := _pDailySched^.nEntrySize + 16#80000000;
			END_IF

			(* update pointer each cycle (even if no day follows!) *)
			_NextDay();
		END_FOR
		(* send data *)
		_i := 13;

	13:
		IF _fbWriteProp.bExecute AND (NOT _fbWriteProp.bBusy) THEN
			(* check result *)
			_fbWriteProp.bExecute := FALSE;
			IF _fbWriteProp.bError THEN
				nErrorId := BACnet_ERR_ADS_Write;
			ELSE
				stWeeklySched.nSet := stWeeklySched.nSet +1;
			END_IF
			_i := 100;
		ELSE
			(* start ADS write *)
			_fbWriteProp.bExecute := TRUE;
		END_IF

	100: (* Done *)
		bDone := (nErrorId = BACnet_ERR_NO_ERROR);
		(* release ADS buffer *)
		stBACnet_AdsBuffer.iLocked := 0;
		(* release data array *)
		stWeeklySched.bBusy := FALSE;
		(* go idle *)
		_i := 0;

END_CASE

(* set error flag *)
bError 	:= nErrorId > BACnet_ERR_NO_ERROR;
bBusy 	:= _i > 0;

ACTION _NextDay:
_bNextDay := ((_pDailySched^.nEntrySize AND 16#80000000) = 16#80000000);
_cbTmpSize := _F_BACnet_AlignedSize(_pDailySched^.nEntrySize AND 16#7FFFFFFF) + SIZEOF(_pDailySched^.nEntrySize) + SIZEOF(_pDailySched^.nRes);
_pDailySched := _pDailySched + _cbTmpSize;
_cbTotalBuf := _cbTotalBuf + _cbTmpSize;
_pOldTimeValue := 0;
END_ACTION

ACTION _NextTimeValue:
_bNextTimeValue := (_pTimeValue^.nEntrySize AND 16#80000000) = 16#80000000;
_cbTmpSize := _F_BACnet_AlignedSize(_pTimeValue^.nEntrySize AND 16#7FFFFFFF) + SIZEOF(_pDailySched^.stListEntry.nEntrySize) + SIZEOF(_pDailySched^.stListEntry.nRes);
_pOldTimeValue := _pTimeValue;
_pTimeValue := _pTimeValue + _cbTmpSize;
END_ACTION

END_FUNCTION_BLOCK

// POUs/BACnet ADS/FB_BACnet_GetDiagInfo
FUNCTION_BLOCK FB_BACnet_GetDiagInfo
VAR_INPUT
	sNetId		: T_AmsNetId;
	bExecute	: BOOL;
	tTimeout	: TIME := BACnet_ADSTimeOut;
END_VAR
VAR_OUTPUT
	bBusy		: BOOL;
	bError		: BOOL;
	nErrID		: UDINT;
	stInfo		: ST_BACnet_Diagnosis;
END_VAR
VAR
	_fbAdsRead	: ADSREAD;
END_VAR

(* call ADS read function to receive info data *)
_fbAdsRead(
	NETID	:= sNetId,
	PORT	:= 16#FFFF, (* ADS port of BACnet device adapter *)
	IDXGRP	:= 16#8000000F,
	IDXOFFS	:= 16#0000,
	LEN		:= SIZEOF(stInfo),
	DESTADDR:= ADR(stInfo),
	READ	:= bExecute,
	TMOUT	:= tTimeout,
	BUSY	=> bBusy,
	ERR		=> bError,
	ERRID	=> nErrID);

END_FUNCTION_BLOCK

// POUs/BACnet ADS/FB_BACnet_NSinkAcknEvent
FUNCTION_BLOCK FB_BACnet_NSinkAcknEvent
VAR_INPUT
	bAcknowledge	: BOOL;
	stAcknEvent		: ST_BACnet_NSinkEvent;
	sMessage		: T_MaxString;
END_VAR
VAR_IN_OUT
	stAdsConn		: ST_BACnet_AdsConnection;
END_VAR
VAR_OUTPUT
	bDone			: BOOL;
	bBusy			: BOOL;
	bError			: BOOL;
	nErrorId		: UINT;
END_VAR
VAR
	_fbAdsWrite		: FW_AdsWrite;
	_i				: INT;
	_rtrigGetSet	: R_TRIG;
	_stNSinkRawData	: ST_BACnet_NotificationSinkEventEntry;
	_stringEncode	: FB_BACnet_StringExtEncode;
	_pChrStringExt	: POINTER TO ST_BACnet_CharacterStringExt;
END_VAR

(*

#define BACNET_STRING_MAXLENGTH    256

typedef struct _EventNotificationRequest
{
      ULONG validFields;
      ULONG processIdentifier;
      BACnetObjectIdentifier initiatingDeviceIdentifier;
      BACnetObjectIdentifier eventObjectIdentifier;
      BACnetTimeStamp timeStamp;
      ULONG notificationClass;
      ULONG priority;
      BACnetEventType eventType;
      CHAR messageText[BACNET_STRING_MAXLENGTH];
      BACnetNotifyType notifyType;
      BOOL ackRequired;
      BACnetEventState fromState;
      BACnetEventState toState;
      PBACnetNotificationParameters pEventValues;
}EventNotificationRequest, *PEventNotificationRequest;

*)

(* ADS write *)
_fbAdsWrite(
	sNetId		:= stAdsConn.sAmsNetId,
	nPort		:= stAdsConn.nAmsPort,
	nIdxGrp		:= BACnet_ADSIGRP_NTFSINK_W_EVENTNTF_ACK_BY_PARAMETER,
	nIdxOffs	:= 0,
	cbWriteLen	:= SIZEOF(_stNSinkRawData) - SIZEOF(_stNSinkRawData._fillBytes00),
	pWriteBuff	:= ADR(_stNSinkRawData.validFields),
	bExecute	:= ,
	tTimeout	:= BACnet_ADSTimeOut,
	bBusy		=> ,
	bError		=> ,
	nErrId		=> );

(* trigger start event *)
_rtrigGetSet(CLK:= bAcknowledge, Q=> );

(* state machine *)
CASE _i OF

	0: (* Idle *)
		IF _rtrigGetSet.Q THEN
			IF (NOT stAdsConn.bValid) THEN
				(* ADS connection not valid *)
				nErrorId := BACnet_ERR_INVALID_ADS_CONN;
			ELSIF (NOT stAdsConn.bNSink) THEN
				(* not a notification sink *)
				nErrorId := BACnet_ERR_ADS_NoNotificationSink;
			ELSE
				nErrorId := BACnet_ERR_NO_ERROR;
				_i := 1;
				(* prepare raw data *)
				MEMSET(destAddr:=ADR(_stNSinkRawData), fillByte:=0, n:=SIZEOF(_stNSinkRawData));
				(* encode message text to UTF-8 *)
				_stringEncode(
					pString			:= ADR(sMessage),
					nSize			:= LEN(sMessage),
					pResultExtStr	:= ADR(_stNSinkRawData.messageText),
					cbResult		:= SIZEOF(_stNSinkRawData.messageText),
					bValid			=> ,
					bOverflow		=> ,
					nLength			=> );
				(* fill flags and other information *)
				_stNSinkRawData.ackRequired := FALSE;
				_stNSinkRawData.eventObjectIdentifier := stAcknEvent.tObjectID;
				_stNSinkRawData.eventType := stAcknEvent.eEventType;
				_stNSinkRawData.fromState := stAcknEvent.eFromState;
				_stNSinkRawData.toState := stAcknEvent.eToState;
				_stNSinkRawData.initiatingDeviceIdentifier := stAcknEvent.nDeviceID;
				_stNSinkRawData.notificationClass := stAcknEvent.nNC;
				_stNSinkRawData.notifyType := BACnetNotifyType_ack_notification;
				_stNSinkRawData.priority := stAcknEvent.nPriotity;
				_stNSinkRawData.processIdentifier := stAcknEvent.nProcessID;
				_stNSinkRawData.timeStamp.stDateTime := stAcknEvent.stDateTime;
				_stNSinkRawData.timeStamp.eType := BACnetTimeStampChoice_dateTime;
			END_IF
			(* reset done flag *)
			bDone := FALSE;
		END_IF
		IF (NOT bAcknowledge) THEN
			nErrorId := BACnet_ERR_NO_ERROR;
			bDone := FALSE;
		END_IF

	(* WRITE *)
	1: (* write data over ADS *)
		IF _fbAdsWrite.bExecute THEN
			IF _fbAdsWrite.bError THEN
				_i := 100;
				nErrorId := BACnet_ERR_ADS_Write;
				_fbAdsWrite.bExecute := FALSE;
			ELSIF (NOT _fbAdsWrite.bBusy) THEN
				(* DONE *)
				_fbAdsWrite.bExecute := FALSE;
				_i := 100;
			END_IF
		ELSE
			_fbAdsWrite.bExecute := TRUE;
		END_IF

	100: (* Done *)
		bDone := (nErrorId = BACnet_ERR_NO_ERROR);
		_i := 0;

END_CASE

(* set error flag *)
bError 	:= nErrorId > BACnet_ERR_NO_ERROR;
bBusy 	:= _i > 0;

END_FUNCTION_BLOCK

// POUs/BACnet Helper/String/FB_BACnet_StringExtEncode
FUNCTION_BLOCK FB_BACnet_StringExtEncode (* convert Windows-1252 to ANSI/UTF-8 BACnet Character String *)
VAR_INPUT
	pString			: POINTER TO T_MaxString; (* pointer to Windows-1252 encoded PLC text *)
	nSize			: INT; (* string length or data size of pText field *)
	pResultExtStr	: POINTER TO ST_BACnet_CharacterStringExt;
	cbResult		: UDINT; (* byte size of result data field *)
END_VAR
VAR_OUTPUT
	bValid			: BOOL;
	bOverflow		: BOOL; (* String length overflow (source string too long) *)
	nLength			: UDINT; (* out string data length in byte *)
END_VAR

(* preset valid to FALSE *)
bOverflow := FALSE;
bValid := TRUE;
(* check pointer *)
IF (pString = 0) OR (pResultExtStr = 0) THEN
	nLength := 0;
	bValid := FALSE;
	RETURN;
END_IF

(* clear string *)
MEMSET(destAddr:=pResultExtStr, fillByte:=0, n:=cbResult);
(* check input size *)
IF (nSize <= 0) THEN
	nLength := 0;

(* convert *)
ELSE
	IF (_F_BACnet_EncodeUTF8(
		pString		:= pString,
		cbString	:= TO_UDINT(nSize),
		pResult		:= pResultExtStr,
		cbResult	:= cbResult,
		nResultLen	:= nLength) > cbResult)
	THEN
		bOverflow	:= TRUE;
		bValid		:= FALSE;
	END_IF
END_IF

END_FUNCTION_BLOCK

// POUs/BACnet Helper/[internal]/_F_BACnet_EncodeUTF8
FUNCTION _F_BACnet_EncodeUTF8 : UDINT (* actually byte length of the result utf-8 string (maybe longer than cbResult; means overflow) *)
VAR_INPUT
	pString		: POINTER TO BYTE; (* pointer to Win1252 string beginning *)
	cbString	: UDINT; (* byte size of string (use SIZEOF - don't use LEN) *)
	pResult		: POINTER TO BYTE; (* pointer to result UTF-8 data area *)
	cbResult	: UDINT; (* byte size of result (use SIZEOF - don't use LEN) *)
END_VAR

VAR
	pBy			: POINTER TO BYTE;
	pByArr		: POINTER TO ARRAY[0..3] OF BYTE;
	nCoded		: UINT;
	bOverflow	: BOOL;
END_VAR
(*All VAR_IN_OUT variables have been moved to the end of the declaration due to compatibility reasons*)
VAR_IN_OUT
	nResultLen	: UDINT; (* final resulting string length (<= cbResult) *)
END_VAR

pBy			:= pString;
pByArr		:= pResult;
bOverflow	:= FALSE;
_F_BACnet_EncodeUTF8 := 0;
nResultLen	:= 0;
(* loop over pString *)
WHILE pBy < (pString + cbString) DO
	IF (pBy^ = 0) THEN EXIT; END_IF
	IF bOverflow OR (_F_BACnet_EncodeUTF8 + 3 > cbResult) THEN
		nCoded := _F_BACnet_Win1252ToUtf8(nW1252:=pBy^, pUtf8:=pByArr, bEval:=TRUE);
		IF (NOT bOverflow) AND (_F_BACnet_EncodeUTF8 + nCoded <= cbResult) THEN
			nCoded := _F_BACnet_Win1252ToUtf8(nW1252:=pBy^, pUtf8:=pByArr, bEval:=FALSE);
		ELSE
			bOverflow := TRUE;
		END_IF
	ELSE
		nCoded := _F_BACnet_Win1252ToUtf8(nW1252:=pBy^, pUtf8:=pByArr, bEval:=FALSE);
	END_IF
	IF (NOT bOverflow) THEN
		pByArr := pByArr + UINT_TO_UDINT(nCoded);
		nResultLen := _F_BACnet_EncodeUTF8 + nCoded;
	END_IF
	_F_BACnet_EncodeUTF8 := _F_BACnet_EncodeUTF8 + nCoded;
	pBy := pBy + 1;
END_WHILE
(* add zero termination if needed *)
IF (nResultLen < cbResult) THEN
	pByArr^[0] := 16#00;
END_IF

END_FUNCTION

// POUs/BACnet Helper/[internal]/_F_BACnet_Win1252ToUtf8
FUNCTION _F_BACnet_Win1252ToUtf8 : UINT(0..3)
VAR_INPUT
	nW1252	: BYTE; (* Win1252 character *)
	pUtf8	: POINTER TO ARRAY[0..2] OF BYTE; (* pointer to target character buffer (utf-8) *)
	bEval	: BOOL; (* TRUE = only evaluate expected coding size (0..3 byte) - but don't write data *)
END_VAR
VAR
	pWord	: POINTER TO ARRAY[0..1] OF BYTE;
	wUCS2	: WORD;
END_VAR
VAR CONSTANT
	cRepl	: BYTE := 16#5F;
END_VAR

(*
	Windows-Codepages
874		Thai
932		Japanisch
936		Vereinfachtes Chinesisch
949		Koreanisch
950		Traditionelles Chinesisch
1250	Mitteleuropäisch
1251	Kyrillisch
1252	Westeuropäisch
1253	Griechisch
1254	Türkisch
1255	Hebräisch
1256	Arabisch
1257	Baltisch
1258	Vietnamesisch
*)
(* check pointer *)
IF (pUtf8 = 0) THEN
	(* null pointer *)
	_F_BACnet_Win1252ToUtf8 := 0;
ELSIF (nW1252 <= 16#7F) THEN
	(* basic latin - 1 byte *)
	IF (NOT bEval) THEN
		pUtf8^[0] := nW1252;
	END_IF
	_F_BACnet_Win1252ToUtf8 := 1;
ELSE
	(* convert to UCS-2 first *)
	wUCS2 := _F_BACnet_Win1252ToUCS2(nW1252:=nW1252, bBE:=FALSE);
	pWord := ADR(wUCS2);
	(* convert used ranges *)
	IF (wUCS2 >= 16#80 AND wUCS2 <= 16#BF) THEN
		(* latin-1 supplement *)
		IF (NOT bEval) THEN
			pUtf8^[0] := 16#C2;
			pUtf8^[1] := pWord^[0];
		END_IF
		_F_BACnet_Win1252ToUtf8 := 2;
	ELSIF (wUCS2 >= 16#C0 AND wUCS2 <= 16#FF) THEN
		(* latin-1 supplement *)
		IF (NOT bEval) THEN
			pUtf8^[0] := 16#C3;
			pUtf8^[1] := pWord^[0] - 16#40;
		END_IF
		_F_BACnet_Win1252ToUtf8 := 2;
	ELSIF (wUCS2 >= 16#140 AND wUCS2 <= 16#17F) THEN
		(* latin extended A *)
		IF (NOT bEval) THEN
			pUtf8^[0] := 16#C5;
			pUtf8^[1] := pWord^[0] + 16#40;
		END_IF
		_F_BACnet_Win1252ToUtf8 := 2;
	ELSIF (wUCS2 >= 16#20A0 AND wUCS2 <= 16#20BF) THEN
		(* currency symbols *)
		IF (NOT bEval) THEN
			pUtf8^[0] := 16#E2;
			pUtf8^[1] := 16#82;
			pUtf8^[2] := pWord^[0];
		END_IF
		_F_BACnet_Win1252ToUtf8 := 3;
	ELSE
		(* unsupported *)
		IF (NOT bEval) THEN
			pUtf8^[0] := cRepl;
		END_IF
		_F_BACnet_Win1252ToUtf8 := 1;
	END_IF
END_IF

END_FUNCTION

// POUs/BACnet Helper/[internal]/_F_BACnet_Win1252ToUCS2
FUNCTION _F_BACnet_Win1252ToUCS2 : WORD
VAR_INPUT
	nW1252 : BYTE;
	bBE	: BOOL; (* byte-order big endian = TRUE *)
END_VAR
VAR
	pArr : POINTER TO ARRAY[0..1] OF BYTE;
	nBuf : BYTE;
	wUCS2: WORD;
END_VAR

(*
	Windows-Codepages
874		Thai
932		Japanisch
936		Vereinfachtes Chinesisch
949		Koreanisch
950		Traditionelles Chinesisch
1250	Mitteleuropäisch
1251	Kyrillisch
1252	Westeuropäisch
1253	Griechisch
1254	Türkisch
1255	Hebräisch
1256	Arabisch
1257	Baltisch
1258	Vietnamesisch
*)
CASE nW1252 OF
	16#9F: wUCS2 := 16#178;
	16#9C: wUCS2 := 16#153;
	16#8C: wUCS2 := 16#152;
	16#9E: wUCS2 := 16#17E;
	16#8E: wUCS2 := 16#17D;
	16#9A: wUCS2 := 16#161;
	16#8A: wUCS2 := 16#160;
	16#80: wUCS2 := 16#20AC;
	ELSE
	wUCS2 := nW1252;
END_CASE
IF bBE THEN
	pArr := ADR(wUCS2);
	nBuf := pArr^[0];
	pArr^[0] := pArr^[1];
	pArr^[1] := nBuf;
END_IF
_F_BACnet_Win1252ToUCS2 := wUCS2;

END_FUNCTION

// POUs/BACnet ADS/FB_BACnet_NSinkReadEvent
FUNCTION_BLOCK FB_BACnet_NSinkReadEvent
VAR_INPUT
	nIndex			: UDINT;
	bAutoGet		: BOOL:=TRUE; (* TRUE = get data when ADS connection or index changed *)
	bGet			: BOOL; (* FALSE --> TRUE = get data from property *)
END_VAR
VAR_IN_OUT
	stAdsConn		: ST_BACnet_AdsConnection;
END_VAR
VAR_OUTPUT
	bDone			: BOOL;
	bNoEntry		: BOOL;
	bBusy			: BOOL;
	bError			: BOOL;
	nErrorId		: UINT;
	stEvent			: ST_BACnet_NSinkEvent;
END_VAR
VAR
	_fbAdsRead		: FW_AdsRead;
	_i				: INT;
	_nOldIndex		: UDINT;
	_rtrigGetSet	: R_TRIG;
	_nAdsReloadOld	: USINT;
	_stNSinkRawData	: ST_BACnet_NotificationSinkEventEntry;
	_StringExtDecode: FB_BACnet_StringExtDecode;
END_VAR

(*

#define BACNET_STRING_MAXLENGTH    256


enum EventNotificationRequestFields
{
      notify_processIdentifier,
      notify_initiatingDeviceIdentifier,
      notify_eventObjectIdentifier,
      notify_timeStamp,
      notify_notificationClass,
      notify_priority,
      notify_eventType,
      notify_messageText,
      notify_notifyType,
      notify_ackRequired,
      notify_fromState,
      notify_toState,
      notify_eventValues,
};

typedef struct _EventNotificationRequest
{
      ULONG validFields;
      ULONG processIdentifier;
      BACnetObjectIdentifier initiatingDeviceIdentifier;
      BACnetObjectIdentifier eventObjectIdentifier;
      BACnetTimeStamp timeStamp;
      ULONG notificationClass;
      ULONG priority;
      BACnetEventType eventType;
      CHAR messageText[BACNET_STRING_MAXLENGTH];
      BACnetNotifyType notifyType;
      BOOL ackRequired;
      BACnetEventState fromState;
      BACnetEventState toState;
      PBACnetNotificationParameters pEventValues;
}EventNotificationRequest, *PEventNotificationRequest;


*)

(* ADS read *)
_fbAdsRead(
	sNetId		:= stAdsConn.sAmsNetId,
	nPort		:= stAdsConn.nAmsPort,
	nIdxGrp		:= BACnet_ADSIGRP_NTFSINK_EVENTNTF_READ,
	nIdxOffs	:= nIndex,
	cbReadLen	:= SIZEOF(_stNSinkRawData),
	pReadBuff	:= ADR(_stNSinkRawData),
	bExecute	:= ,
	tTimeout	:= BACnet_ADSTimeOut,
	bBusy		=> ,
	bError		=> ,
	nErrId		=> ,
	cbRead		=> );

(* trigger start event *)
_rtrigGetSet(CLK:= bGet, Q=> );

(* state machine *)
CASE _i OF

	0: (* Idle *)
		IF		(		(		_rtrigGetSet.Q
							OR	(_nAdsReloadOld <> stAdsConn.nReload)
							OR	(_nOldIndex <> nIndex)
						)
					AND	bAutoGet
				)
			OR	_rtrigGetSet.Q
		THEN
			IF (NOT stAdsConn.bValid) THEN
				(* ADS connection not valid *)
				nErrorId := BACnet_ERR_INVALID_ADS_CONN;
			ELSIF (NOT stAdsConn.bNSink) THEN
				(* not a notification sink *)
				nErrorId := BACnet_ERR_ADS_NoNotificationSink;
			ELSE
				nErrorId := BACnet_ERR_NO_ERROR;
				_i := 1;
				MEMSET(destAddr:=ADR(_stNSinkRawData), fillByte:=0, n:=SIZEOF(_stNSinkRawData));
				(* remind ADS reload counter and parameter *)
				_nAdsReloadOld := stAdsConn.nReload;
				_nOldIndex := nIndex;
			END_IF
			(* reset done flag *)
			bDone := FALSE;
			bNoEntry := FALSE;
		END_IF
		IF (NOT bGet) AND (NOT bAutoGet) THEN
			nErrorId := BACnet_ERR_NO_ERROR;
			bDone := FALSE;
		END_IF

	(* READ *)
	1: (* read data over ADS *)
		IF _fbAdsRead.bExecute THEN
			IF _fbAdsRead.bError THEN
				_i := 100;
				(* entry exists? *)
				bNoEntry := ((UDINT_TO_DWORD(_fbAdsRead.nErrId) AND 16#FFF) = 16#703);
				IF (NOT bNoEntry) THEN
					nErrorId := BACnet_ERR_ADS_Read;
				END_IF
				_fbAdsRead.bExecute := FALSE;
			ELSIF (NOT _fbAdsRead.bBusy) THEN
				_fbAdsRead.bExecute := FALSE;
				(* check size *)
				IF (_fbAdsRead.cbRead < 312) THEN
					(* wrong data size *)
					nErrorId := BACnet_ERR_ADS_Data;
				ELSE
					(* get the valid fields info *)
					stEvent.stValidFields.bProcessIdentifier			:= _stNSinkRawData.validFields.0;
					stEvent.stValidFields.bInitiatingDeviceIdentifier	:= _stNSinkRawData.validFields.1;
					stEvent.stValidFields.bEventObjectIdentifier		:= _stNSinkRawData.validFields.2;
					stEvent.stValidFields.bTimeStamp					:= _stNSinkRawData.validFields.3;
					stEvent.stValidFields.bNotificationClass			:= _stNSinkRawData.validFields.4;
					stEvent.stValidFields.bPriority						:= _stNSinkRawData.validFields.5;
					stEvent.stValidFields.bEventType					:= _stNSinkRawData.validFields.6;
					stEvent.stValidFields.bMessageText					:= _stNSinkRawData.validFields.7;
					stEvent.stValidFields.bNotifyType					:= _stNSinkRawData.validFields.8;
					stEvent.stValidFields.bAckRequired					:= _stNSinkRawData.validFields.9;
					stEvent.stValidFields.bFromState					:= _stNSinkRawData.validFields.10;
					stEvent.stValidFields.bToState						:= _stNSinkRawData.validFields.11;
					stEvent.stValidFields.bEventValues					:= _stNSinkRawData.validFields.12;
					(* copy data according to event valid flags *)
					IF (stEvent.stValidFields.bAckRequired) THEN
						stEvent.bAcknReq := _stNSinkRawData.ackRequired;
					END_IF
					IF (stEvent.stValidFields.bEventType) THEN
						stEvent.eEventType := _stNSinkRawData.eventType;
					END_IF
					IF (stEvent.stValidFields.bFromState) THEN
						stEvent.eFromState := _stNSinkRawData.fromState;
					END_IF
					IF (stEvent.stValidFields.bNotifyType) THEN
						stEvent.eNotifyType := _stNSinkRawData.notifyType;
					END_IF
					IF (stEvent.stValidFields.bToState) THEN
						stEvent.eToState := _stNSinkRawData.toState;
					END_IF
					IF (stEvent.stValidFields.bInitiatingDeviceIdentifier) THEN
						stEvent.nDeviceID := _stNSinkRawData.initiatingDeviceIdentifier;
					END_IF
					IF (stEvent.stValidFields.bNotificationClass) THEN
						stEvent.nNC := _stNSinkRawData.notificationClass;
					END_IF
					IF (stEvent.stValidFields.bPriority) THEN
						stEvent.nPriotity := _stNSinkRawData.priority;
					END_IF
					IF (stEvent.stValidFields.bProcessIdentifier) THEN
						stEvent.nProcessID := _stNSinkRawData.processIdentifier;
					END_IF
					IF (		stEvent.stValidFields.bTimeStamp
							AND	(_stNSinkRawData.timeStamp.eType = BACnetTimeStampChoice_dateTime))
					THEN
						stEvent.stDateTime := _stNSinkRawData.timeStamp.stDateTime;
					ELSE
						stEvent.stDateTime.stDate.nDay := 16#FF;
						stEvent.stDateTime.stDate.nDayOfWeek := 16#FF;
						stEvent.stDateTime.stDate.nMonth := 16#FF;
						stEvent.stDateTime.stDate.nYear := 16#FF;
						stEvent.stDateTime.stTime.nHour := 16#FF;
						stEvent.stDateTime.stTime.nMinute := 16#FF;
						stEvent.stDateTime.stTime.nSecond := 16#FF;
						stEvent.stDateTime.stTime.nHundredths := 16#FF;
					END_IF
					IF (stEvent.stValidFields.bEventObjectIdentifier) THEN
						stEvent.tObjectID := _stNSinkRawData.eventObjectIdentifier;
					END_IF
					IF (stEvent.stValidFields.bMessageText) THEN
						(* decode message text *)
						_StringExtDecode(
							pChrStringExt	:= ADR(_stNSinkRawData.messageText),
							cbOutSize		:= MIN(SIZEOF(_stNSinkRawData.messageText), SIZEOF(stEvent.sMessage)),
							pOutString		:= ADR(stEvent.sMessage),
							bValid			=> ,
							bOverflow		=> ,
							nLength			=> ,
							eSrcEncoding	=> );

						(* check overflow flag *)
						IF _StringExtDecode.bOverflow THEN
							nErrorId := BACnet_ERR_ADS_BufferSize;
	
						(* check encoding supported flag *)
						ELSIF (NOT _StringExtDecode.bValid) THEN
							nErrorId := BACnet_ERR_ADS_Encoding;
						END_IF
					END_IF

				END_IF
				(* DONE *)
				_i := 100;
			END_IF
		ELSE
			MEMSET(destAddr:=ADR(stEvent), fillByte:=0, n:=SIZEOF(stEvent));
			_fbAdsRead.bExecute := TRUE;
		END_IF

	100: (* Done *)
		bDone := (nErrorId = BACnet_ERR_NO_ERROR) AND (NOT bNoEntry);
		_i := 0;

END_CASE

(* set error flag *)
bError 	:= nErrorId > BACnet_ERR_NO_ERROR;
bBusy 	:= _i > 0;

END_FUNCTION_BLOCK

// POUs/BACnet ADS/FB_BACnet_NSinkRemoveEvent
FUNCTION_BLOCK FB_BACnet_NSinkRemoveEvent
VAR_INPUT
	bRemove		: BOOL;
	nIndex		: UDINT;
END_VAR
VAR_IN_OUT
	stAdsConn	: ST_BACnet_AdsConnection;
END_VAR
VAR_OUTPUT
	bDone		: BOOL;
	bNoEntry	: BOOL;
	bBusy		: BOOL;
	bError		: BOOL;
	nErrorId	: UINT;
END_VAR
VAR
	_fbAdsRead	: FW_AdsRead;
	_i			: INT;
	_rtrigGetSet: R_TRIG;
END_VAR

(* ADS read *)
_fbAdsRead(
	sNetId		:= stAdsConn.sAmsNetId,
	nPort		:= stAdsConn.nAmsPort,
	nIdxGrp		:= BACnet_ADSIGRP_NTFSINK_EVENTNTF_DELETE,
	nIdxOffs	:= nIndex,
	cbReadLen	:= 0,
	pReadBuff	:= 0,
	bExecute	:= ,
	tTimeout	:= BACnet_ADSTimeOut,
	bBusy		=> ,
	bError		=> ,
	nErrId		=> ,
	cbRead		=> );

(* trigger start event *)
_rtrigGetSet(CLK:= bRemove, Q=> );

(* state machine *)
CASE _i OF

	0: (* Idle *)
		IF _rtrigGetSet.Q THEN
			IF (NOT stAdsConn.bValid) THEN
				(* ADS connection not valid *)
				nErrorId := BACnet_ERR_INVALID_ADS_CONN;
			ELSIF (NOT stAdsConn.bNSink) THEN
				(* not a notification sink *)
				nErrorId := BACnet_ERR_ADS_NoNotificationSink;
			ELSE
				nErrorId := BACnet_ERR_NO_ERROR;
				_i := 1;
			END_IF
			(* reset done flag *)
			bDone := FALSE;
			(* reset no-entry flag *)
			bNoEntry := FALSE;
		END_IF
		IF (NOT bRemove) THEN
			nErrorId := BACnet_ERR_NO_ERROR;
			bDone := FALSE;
		END_IF

	(* READ *)
	1: (* read object property data over ADS *)
		IF _fbAdsRead.bExecute THEN
			IF _fbAdsRead.bError THEN
				_i := 100;
				(* entry exists? *)
				bNoEntry := ((UDINT_TO_DWORD(_fbAdsRead.nErrId) AND 16#FFF) = 16#703);
				IF (NOT bNoEntry) THEN
					nErrorId := BACnet_ERR_ADS_Read;
				END_IF
				_fbAdsRead.bExecute := FALSE;
			ELSIF (NOT _fbAdsRead.bBusy) THEN
				_fbAdsRead.bExecute := FALSE;
				(* DONE *)
				_i := 100;
			END_IF
		ELSE
			_fbAdsRead.bExecute := TRUE;
		END_IF

	100: (* Done *)
		bDone := (nErrorId = BACnet_ERR_NO_ERROR) AND (NOT bNoEntry);
		_i := 0;

END_CASE

(* set error flag *)
bError 	:= nErrorId > BACnet_ERR_NO_ERROR;
bBusy 	:= _i > 0;

END_FUNCTION_BLOCK

// POUs/BACnet ADS/FB_BACnet_TimeSync
FUNCTION_BLOCK FB_BACnet_TimeSync
VAR_INPUT
	bExecute	: BOOL; (* Synchronize BACnet time information with local system time and, if set, send broadcast message *)
	bBroadcast	: BOOL := TRUE; (* Synchronize BACnet with broadcast message (FALSE = No broadcast [Rev-12-only feature]) *)
	tTimeout	: TIME := BACnet_ADSTimeOut;
END_VAR
VAR_IN_OUT
	Device		: FB_BACnet_Device;
END_VAR
VAR_OUTPUT
	bReady		: BOOL; (* local time information is valid *)
	bBusy		: BOOL;
	bError		: BOOL;
	nErrID		: UDINT;
	tsSystemTime: TIMESTRUCT; (* local system time (windows time) as TIMESTRUCT *)
	dtSystemTime: ST_BACnet_DateTime; (* local system time (windows time) as BACnet_Date_Time *)
	tzID		: E_TimeZoneID;
	tzInfo		: ST_TimeZoneInformation;
	tsUTC		: TIMESTRUCT; (* UTC system time (GMT) *)
END_VAR
VAR
	_fbAdsWrite	: ADSWRITE;
	_fbLocalTime: FB_LocalSystemTime;
	_fbGetTzInfo: FB_GetTimeZoneInformation;
	_fbUTC		: FB_TzSpecificLocalTimeToSystemTime;
	_oldTzId	: E_TimeZoneID := eTimeZoneID_Invalid;
	_tofReload	: TOF;
	_dtUTC		: ST_BACnet_DateTime;
END_VAR

(* read local time *)
_fbLocalTime(
	sNetID	:= '',
	bEnable	:= TRUE,
	dwCycle	:= ,
	dwOpt	:= ,
	tTimeout:= tTimeout,
	bValid	=> ,
	systemTime=> tsSystemTime,
	tzID	=> );

_fbGetTzInfo(
	sNetID	:= '',
	bExecute:= _fbLocalTime.bValid AND (_oldTzId <> _fbLocalTime.tzID) AND (NOT _tofReload.Q),
	tTimeout:= tTimeout,
	bBusy	=> ,
	bError	=> ,
	nErrID	=> ,
	tzID	=> ,
	tzInfo	=> tzInfo);

_tofReload(
	IN	:= _fbGetTzInfo.bError AND (NOT _tofReload.Q),
	PT	:= tTimeout,
	Q	=> ,
	ET	=> );

IF _fbGetTzInfo.bExecute AND (NOT _fbGetTzInfo.bBusy) THEN
	IF (NOT _fbGetTzInfo.bError) THEN
		_oldTzId := _fbLocalTime.tzID;
	ELSE
		_oldTzId := eTimeZoneID_Invalid;
	END_IF
END_IF

_fbUTC(
	in		:= _fbLocalTime.systemTime,
	tzInfo	:= _fbGetTzInfo.tzInfo,
	out		=> tsUTC,
	eTzID	=> tzID,
	bB		=> );

(* check if all information are valid *)
bReady := _fbLocalTime.bValid AND (NOT _fbGetTzInfo.bError) AND (_fbUTC.eTzID > eTimeZoneID_Unknown) AND Device.stAdsConn.bValid;

(* convert to BACnet_Date_Time *)
dtSystemTime:= F_BACnet_TimeStruct_TO_DateTime(tsSystemTime);
_dtUTC		:= F_BACnet_TimeStruct_TO_DateTime(tsUTC);

(* call ADS write function to synchronize system time *)
IF bBroadcast THEN
	_fbAdsWrite.IDXOFFS	:= 16#0000;
ELSE
	_fbAdsWrite.IDXOFFS	:= 16#0001;
END_IF
_fbAdsWrite(
	NETID	:= Device.stAdsConn.sAmsNetId,
	PORT	:= 16#FFFF, (* AMS port of BACnet device adapter *)
	IDXGRP	:= 16#8000002D,
	LEN		:= SIZEOF(_dtUTC),
	SRCADDR	:= ADR(_dtUTC),
	WRITE	:= bReady AND bExecute,
	TMOUT	:= tTimeout,
	BUSY	=> bBusy,
	ERR		=> bError,
	ERRID	=> nErrID);

END_FUNCTION_BLOCK

// POUs/BACnet Helper/DateTime/F_BACnet_TimeStruct_TO_DateTime
FUNCTION F_BACnet_TimeStruct_TO_DateTime : ST_BACnet_DateTime
VAR_INPUT
	IN	: TIMESTRUCT;
END_VAR

F_BACnet_TimeStruct_TO_DateTime.stDate.nDay			:= WORD_TO_BYTE(IN.wDay);
IF IN.wDayOfWeek = 0 THEN
	F_BACnet_TimeStruct_TO_DateTime.stDate.nDayOfWeek := 7;
ELSE
	F_BACnet_TimeStruct_TO_DateTime.stDate.nDayOfWeek := WORD_TO_BYTE(IN.wDayOfWeek);
END_IF
F_BACnet_TimeStruct_TO_DateTime.stDate.nMonth		:= WORD_TO_BYTE(IN.wMonth);
F_BACnet_TimeStruct_TO_DateTime.stDate.nYear		:= WORD_TO_BYTE(IN.wYear - 1900);
F_BACnet_TimeStruct_TO_DateTime.stTime.nHour		:= WORD_TO_BYTE(IN.wHour);
F_BACnet_TimeStruct_TO_DateTime.stTime.nMinute		:= WORD_TO_BYTE(IN.wMinute);
F_BACnet_TimeStruct_TO_DateTime.stTime.nSecond		:= WORD_TO_BYTE(IN.wSecond);
F_BACnet_TimeStruct_TO_DateTime.stTime.nHundredths	:= WORD_TO_BYTE(IN.wMilliseconds / 10);

END_FUNCTION

// POUs/BACnet Helper/[internal]/_F_BACnet_SetBitFieldBit
FUNCTION _F_BACnet_SetBitFieldBit : DWORD
VAR_INPUT
	ptrData		:	POINTER TO DWORD;
	bitNbr			:	INT;
END_VAR
VAR
END_VAR

ptrData^ := ptrData^ OR (SHR(DWORD#16#00008000, _F_BACnet_BitFieldBit(bitNbr)));
_F_BACnet_SetBitFieldBit := ptrData^;

END_FUNCTION

// POUs/BACnet Helper/[internal]/_F_BACnet_UnSetBitFieldBit
FUNCTION _F_BACnet_UnSetBitFieldBit : DWORD
VAR_INPUT
	ptrData		:	POINTER TO DWORD;
	bitNbr			:	INT;
END_VAR
VAR
END_VAR

ptrData^ := ptrData^ AND NOT (SHR(DWORD#16#00008000,_F_BACnet_BitFieldBit(bitNbr)));
_F_BACnet_UnSetBitFieldBit := ptrData^;

END_FUNCTION

// POUs/BACnet Helper/[internal]/_FB_BACnet_PidTune
FUNCTION_BLOCK _FB_BACnet_PidTune
VAR_INPUT
	bStart	: BOOL;
	bStop	: BOOL; (* Abort tuning process *)
	fSetY	: REAL;
	fX		: REAL;
	fDeadband	: REAL;
	tTimeout: TIME := T#15m;
	fMinY	: REAL;
	fMaxY	: REAL;
	fCycleTime : REAL; (* cycle time in seconds [s]; 0 = use internal measuring *)
	eMode	: E_BACNETPIDTUNINGMODE := BACnetPIDTuningMode_PI;
END_VAR
VAR_IN_OUT
	fY		: REAL;
END_VAR
VAR_OUTPUT
	fPID_Kp	: REAL;
	fPID_Ki	: REAL;
	fPID_Kd	: REAL;
	eAction	: E_BACNETACTION;
	bSetY	: BOOL;
	bWaitY	: BOOL;
	bWaitX	: BOOL;
	bReady	: BOOL;
	bBusy	: BOOL;
	bDone	: BOOL;
	bAborted: BOOL;
	bTimeout: BOOL;
END_VAR
VAR
	_oldY	: REAL;
	_fbPT1_D: FB_BACnet_PT1;
	_step : INT;
	_sysTime	: GETCPUCOUNTER;
	_Time : T_LARGE_INTEGER;
	_TimeOld : T_LARGE_INTEGER;
	_TimeStart : T_LARGE_INTEGER;
	_fbAvg : FB_BACnet_AvgValue;
	_fCycleTime : REAL;
	_oldX : REAL;
	_highest : ARRAY[0..9] OF ARRAY[0..1] OF REAL;
	_HighestPoint : ARRAY[0..1] OF REAL;
	_nFifoHigh : INT;
	_nFifoCount : DINT;
	_fDsum : REAL;
	_fDhigh : REAL;
	_tonTimeout : TON;
	_tofYRemain : TOF;
	_tofXRemain : TOF;
	_StartPoint : ARRAY[0..1] OF REAL;
	_EndPoint : ARRAY[0..1] OF REAL;
	_fn : REAL;
	_fTu : REAL;
	_fPID_Tn : REAL;
	_fPID_Tv : REAL;
	_tonStartDelay : TON;
	_fStartX : REAL;
	_fStartY : REAL;
	_tonMeasureTrigger : TON;
	_Xp : REAL;
	_D	: REAL;
	_bDsink : BOOL;
	_bMinScanTime : BOOL;
END_VAR

_tofYRemain(IN:= (fY <> _oldY), PT:= (tTimeout / 100), Q=> , ET=> );
_tofXRemain(IN:= (ABS(_fbPT1_D.Y) > ABS(fDeadband)), PT:= (tTimeout / 100), Q=> , ET=> );

(* timeout *)
_tonTimeout(IN:= , PT:= tTimeout, Q=> , ET=> );

(* record exact cycle time *)
_TimeOld := _Time;
_sysTime(
	cpuCntLoDW=> _Time.dwLowPart,
	cpuCntHiDW=> _Time.dwHighPart);

(* average filter for input value *)
_fbAvg(X:= fX, n:= 100, Y=> );
(* trigger timer *)
_tonMeasureTrigger(IN:= NOT _tonMeasureTrigger.Q, PT:= (tTimeout / 300), Q=> , ET=> );
(* calculate gradient on trigger event *)
IF _tonMeasureTrigger.Q THEN
	_fCycleTime := _F_BACnet_SysTimeDiff(_Time, _TimeOld); (* [s] *)
	IF (_fCycleTime > 0.0) THEN
		(* calculate gradient *)
		_D := (_fbAvg.Y - _oldX) / _fCycleTime;
	END_IF
	(* reset average filter *)
	_fbAvg(X:= _fbAvg.Y, n:= 0, Y=> );
	(* reset trigger *)
	_tonMeasureTrigger(IN := FALSE);
END_IF
(* gradient filter *)
_fbPT1_D(X:= _D, T:= TIME_TO_REAL(tTimeout) / 1000.0 / 200.0, Tcycle:= fCycleTime, Y=> );

bWaitX := _tofXRemain.Q AND (_step = 0);
bWaitY := _tofYRemain.Q AND (_step = 0);
bReady :=	(NOT bWaitX)
		AND	(NOT bWaitY)
		AND (_step = 0);
_tonStartDelay(IN:= bStart AND bReady, PT:= (tTimeout / 100), Q=> , ET=> );

bSetY := FALSE;

CASE _step OF

	0:
		IF bStart AND (NOT bStop) THEN
			IF _tonStartDelay.Q THEN
				bReady := FALSE;
				_StartPoint[0] := 0.0;
				_StartPoint[1] := fX;
				_step := 10;
				_TimeStart := _Time;
				_fStartY := fY;
				_fStartX := fX;
				_tonTimeout.IN := FALSE;
			ELSE
				_tonTimeout.IN := TRUE;
			END_IF
		ELSE
			bWaitY := FALSE;
			bWaitX := FALSE;
			_tonTimeout.IN := FALSE;
		END_IF

	10: (* wait start condition *)
		fY := fSetY;
		bWaitX := TRUE;
		bSetY := TRUE;
		_tonTimeout.IN := TRUE;
		IF bStop THEN
			_step := 200;
		ELSIF (_tonTimeout.Q) THEN
			_step := 200;
		ELSIF	(_fbAvg.Y > _fStartX + ABS(fDeadband))
			OR	(_fbAvg.Y < _fStartX - ABS(fDeadband))
		THEN
			_step := 20;
			_nFifoHigh := 0;
			_fDhigh := 0.0;
			_nFifoCount := 0;
			_fDsum := 0.0;
			_tonTimeout.IN := FALSE;
		END_IF

	20: (* record *)
		bWaitX := TRUE;
		bSetY := TRUE;
		_tonTimeout.IN := TRUE;
		IF bStop THEN
			_step := 200;
		ELSIF _tonTimeout.Q THEN
			_step := 200;
			bTimeout := TRUE;
		ELSIF	((_D > _fDhigh) AND (_fbAvg.Y > _fStartX)) (* direct system / pos. acceleration *)
			OR	((_D < _fDhigh) AND (_fbAvg.Y < _fStartX)) (* reverse system / neg. acceleration *)
		THEN
			_fDsum := _fDsum + _fbPT1_D.Y;
			IF (_nFifoCount >= 10) THEN
				_fDsum := _fDsum - _highest[_nFifoHigh][1];
			END_IF
			(* remind highest gradiant *)
			_fDhigh := _D;
			(* fill into FIFO *)
			_highest[_nFifoHigh][0] := _F_BACnet_SysTimeDiff(_Time, _TimeStart);
			_highest[_nFifoHigh][1] := _fbPT1_D.Y;
			(* remind highest point *)
			_HighestPoint[0] := _highest[_nFifoHigh][0];	(* t [s] *)
			_HighestPoint[1] := _fbAvg.Y;							(* X [1] *)
			(* count FIFO position and counter *)
			_nFifoHigh := (_nFifoHigh + 1) MOD 10;
			_nFifoCount := _nFifoCount + 1;
		END_IF
		(* check scan time *)
		_bMinScanTime := (_F_BACnet_SysTimeDiff(_Time, _TimeStart) >= ((TIME_TO_REAL(tTimeout) / 1000.0) / 10.0));
		(* exit, when acceleration sinks *)
		IF		(_nFifoCount >= 10)
			AND	_bMinScanTime
		THEN
			(* sink detected, when gradient fells beneath 30% of averaged gradient *)
			_bDsink := (ABS(_fbPT1_D.Y) <= (ABS(_fDsum / 10.0) * 0.3));
		ELSE
			_bDsink := FALSE;
		END_IF
		IF 		_bDsink
			OR	(		_bMinScanTime
					AND	(ABS(_fbPT1_D.Y) < (ABS(_fDhigh) * 0.1)) (* less 10% of max. gradient *)
					AND	(_nFifoCount > 1)
				)
		THEN
			_step := 90;
			_EndPoint[0] := _F_BACnet_SysTimeDiff(_Time, _TimeStart);
			_EndPoint[1] := fX;
			_tonTimeout.IN := FALSE;
		END_IF

	90:
		_step := 100;
		fY := _fStartY;

		IF (_fDhigh <> 0.0) AND (fSetY - _fStartY <> 0.0) THEN
			(* calculate linear function offset *)
			_fn := _HighestPoint[1] - (_fDhigh * _HighestPoint[0]);

			(* calculate X intersection with minimum value (Tu)
				Tu = (Ymin - N) / D			 	*)
			_fTu := ABS((_StartPoint[1] - _fn) / _fDhigh);

			IF (_fTu > 0.0) THEN
				(* calculate Kp *)
				_Xp := _fDhigh * _fTu * (fMaxY - fMinY) / (fSetY - _fStartY);
				IF (_Xp >= 0.0) THEN
					eAction := BACnetAction_direct;
				ELSE
					eAction := BACnetAction_reverse;
				END_IF
				_Xp := ABS(_Xp);

				(* decide between tuning modes *)
				CASE eMode OF
					BACnetPIDTuningMode_P:
						(* calculate P controller *)
						_fPID_Tn := 0.0;
						_fPID_Tv := 0.0;
						fPID_Kp := _Xp;
						fPID_Ki := 0.0;
						fPID_Kd := 0.0;

					BACnetPIDTuningMode_PI:
						(* calculate PI controller *)
						_fPID_Tn := 3.3 * _fTu;
						_fPID_Tv := 0.0;
						fPID_Kp := 1.2 * _Xp;
						fPID_Ki := (1 / _fPID_Tn) * fPID_Kp;
						fPID_Kd := 0.0;

					BACnetPIDTuningMode_PD:
						(* calculate PI controller *)
						_fPID_Tn := 0.0;
						_fPID_Tv := 0.25 * _fTu;
						fPID_Kp := 0.83 * _Xp;
						fPID_Ki := 0.0;
						fPID_Kd := _fPID_Tv * fPID_Kp;

					BACnetPIDTuningMode_PID:
						(* calculate PID controller *)
						_fPID_Tn := 2.0 * _fTu;
						_fPID_Tv := 0.5 * _fTu;
						fPID_Kp := 0.83 * _Xp;
						IF (_fPID_Tn <> 0.0) THEN
							fPID_Ki := (1 / _fPID_Tn) * fPID_Kp;
						ELSE
							fPID_Ki := 0.0;
						END_IF
						fPID_Kd := _fPID_Tv * fPID_Kp;

				END_CASE
			ELSE
				_step := 200;
			END_IF
		ELSE
			_step := 200;
		END_IF


	100:
		IF (NOT bStart) THEN
			_step := 0;
		END_IF

	200:
		fY := _fStartY;
		_tonTimeout.IN := FALSE;
		IF (NOT bStart) THEN
			_step := 0;
			bTimeout := FALSE;
		END_IF

END_CASE

bAborted := _step = 200;
bDone := _step = 100;
bBusy := _step > 0 AND (NOT bDone) AND (NOT bAborted);

_oldY := fY;
_oldX := _fbAvg.Y;

END_FUNCTION_BLOCK

// POUs/BACnet Helper/FB_BACnet_AvgValue
FUNCTION_BLOCK FB_BACnet_AvgValue
VAR_INPUT
	X	: REAL; (* input value to average *)
	n	: UINT; (* number of averages (0 = no average --> Y = X) *)
END_VAR
VAR_OUTPUT
	Y	: REAL; (* average result *)
END_VAR
VAR
	_n	: UINT := 0;
	_Xn : LREAL;
END_VAR

IF (_n > n) THEN
	_n := n;
END_IF
IF (_n = 0) OR (n = 0) THEN
	_Xn := REAL_TO_LREAL(X);
ELSE
	_Xn := ((_Xn * _n) + REAL_TO_LREAL(X)) / UINT_TO_LREAL(_n + 1);
END_IF
_n := _n + 1;
Y := LREAL_TO_REAL(_Xn);

END_FUNCTION_BLOCK

// POUs/BACnet Helper/DateTime/F_BACnet_CheckWeekOfMonth
FUNCTION F_BACnet_CheckWeekOfMonth : USINT

VAR
END_VAR
(*All VAR_IN_OUT variables have been moved to the end of the declaration due to compatibility reasons*)
VAR_IN_OUT
	nIn	: BYTE;
END_VAR

IF nIn > 7 OR nIn = 0 THEN
	F_BACnet_CheckWeekOfMonth := 255;
ELSE
	F_BACnet_CheckWeekOfMonth := nIn;
END_IF
nIn := F_BACnet_CheckWeekOfMonth;

END_FUNCTION

// POUs/BACnet Helper/DateTime/F_BACnet_DateHasPlaceholder
FUNCTION F_BACnet_DateHasPlaceholder : BOOL
VAR_INPUT
	stDate		: ST_BACnet_Date;
END_VAR

F_BACnet_DateHasPlaceholder := (stDate.nDay = 16#FF) OR (stDate.nDayOfWeek = 16#FF) OR (stDate.nMonth = 16#FF) OR (stDate.nYear = 16#FF);

END_FUNCTION

// POUs/BACnet Helper/DateTime/F_BACnet_DateTime_TO_TimeStruct
FUNCTION F_BACnet_DateTime_TO_TimeStruct : TIMESTRUCT
VAR_INPUT
	IN	: ST_BACnet_DateTime;
END_VAR

F_BACnet_DateTime_TO_TimeStruct.wDay			:= BYTE_TO_WORD(IN.stDate.nDay);
F_BACnet_DateTime_TO_TimeStruct.wDayOfWeek		:= BYTE_TO_WORD(IN.stDate.nDayOfWeek MOD 7);
F_BACnet_DateTime_TO_TimeStruct.wDay			:= BYTE_TO_WORD(IN.stDate.nDay);
F_BACnet_DateTime_TO_TimeStruct.wMonth			:= BYTE_TO_WORD(IN.stDate.nMonth);
F_BACnet_DateTime_TO_TimeStruct.wYear			:= BYTE_TO_WORD(IN.stDate.nYear) + 1900;
F_BACnet_DateTime_TO_TimeStruct.wHour			:= BYTE_TO_WORD(IN.stTime.nHour);
F_BACnet_DateTime_TO_TimeStruct.wMinute			:= BYTE_TO_WORD(IN.stTime.nMinute);
F_BACnet_DateTime_TO_TimeStruct.wSecond			:= BYTE_TO_WORD(IN.stTime.nSecond);
F_BACnet_DateTime_TO_TimeStruct.wMilliseconds	:= BYTE_TO_WORD(IN.stTime.nHundredths) * 10;

END_FUNCTION

// POUs/BACnet Helper/DateTime/F_BACnet_DateTimeString
FUNCTION F_BACnet_DateTimeString : STRING(19)

VAR
	str : STRING;
END_VAR
(*All VAR_IN_OUT variables have been moved to the end of the declaration due to compatibility reasons*)
VAR_IN_OUT
	stDateTime		: ST_BACnet_DateTime;
END_VAR

str := '';
IF stDateTime.stDate.nDay >= 1 THEN
	IF stDateTime.stDate.nDay <= 9 THEN
		str := CONCAT(str, CONCAT('0', BYTE_TO_STRING(stDateTime.stDate.nDay)));
	ELSIF stDateTime.stDate.nDay <= 31 THEN
		str := CONCAT(str, BYTE_TO_STRING(stDateTime.stDate.nDay));
	ELSE
		str := CONCAT(str, '**');
	END_IF
ELSE
	str := CONCAT(str, '**');
END_IF

str := CONCAT(str, '.');
IF stDateTime.stDate.nMonth >= 1 THEN
	IF stDateTime.stDate.nMonth <= 9 THEN
		str := CONCAT(str, CONCAT('0', BYTE_TO_STRING(stDateTime.stDate.nMonth)));
	ELSIF stDateTime.stDate.nMonth <= 12 THEN
		str := CONCAT(str, BYTE_TO_STRING(stDateTime.stDate.nMonth));
	ELSE
		str := CONCAT(str, '**');
	END_IF
ELSE
	str := CONCAT(str, '**');
END_IF

str := CONCAT(str, '.');
IF stDateTime.stDate.nYear < 16#FF THEN
	str := CONCAT(str, UINT_TO_STRING(BYTE_TO_UINT(stDateTime.stDate.nYear) + 1900));
ELSE
	str := CONCAT(str, '****');
END_IF

str := CONCAT(str, ' ');
str := CONCAT(str, F_BACnet_TimeString(stDateTime.stTime));
F_BACnet_DateTimeString := str;

END_FUNCTION

// POUs/BACnet Helper/DateTime/F_BACnet_TimeString
FUNCTION F_BACnet_TimeString : STRING(12)

VAR
	str : STRING;
END_VAR
(*All VAR_IN_OUT variables have been moved to the end of the declaration due to compatibility reasons*)
VAR_IN_OUT
	stTime : ST_BACnet_Time;
END_VAR

str := '';
IF stTime.nHour <= 9 THEN
	str := CONCAT(str, CONCAT('0', BYTE_TO_STRING(stTime.nHour)));
ELSIF stTime.nHour <= 23 THEN
	str := CONCAT(str, BYTE_TO_STRING(stTime.nHour));
ELSE
	str := CONCAT(str, '**');
END_IF

str := CONCAT(str, ':');
IF stTime.nMinute <= 9 THEN
	str := CONCAT(str, CONCAT('0', BYTE_TO_STRING(stTime.nMinute)));
ELSIF stTime.nMinute <= 59 THEN
	str := CONCAT(str, BYTE_TO_STRING(stTime.nMinute));
ELSE
	str := CONCAT(str, '**');
END_IF

str := CONCAT(str, ':');
IF stTime.nSecond <= 9 THEN
	str := CONCAT(str, CONCAT('0', BYTE_TO_STRING(stTime.nSecond)));
ELSIF stTime.nSecond <= 59 THEN
	str := CONCAT(str, BYTE_TO_STRING(stTime.nSecond));
ELSE
	str := CONCAT(str, '**');
END_IF

str := CONCAT(str, '.');
IF stTime.nHundredths <= 9 THEN
	str := CONCAT(str, CONCAT('0', BYTE_TO_STRING(stTime.nHundredths)));
ELSIF stTime.nHundredths <= 99 THEN
	str := CONCAT(str, BYTE_TO_STRING(stTime.nHundredths));
ELSE
	str := CONCAT(str, '**');
END_IF
F_BACnet_TimeString := str;

END_FUNCTION

// POUs/BACnet Helper/DateTime/F_BACnet_TimeHasPlaceholder
FUNCTION F_BACnet_TimeHasPlaceholder : BOOL
VAR_INPUT
	stTime		: ST_BACnet_Time;
END_VAR

F_BACnet_TimeHasPlaceholder := (stTime.nHour = 16#FF) OR (stTime.nHundredths = 16#FF) OR (stTime.nMinute = 16#FF) OR (stTime.nSecond = 16#FF);

END_FUNCTION

// POUs/BACnet Helper/Flags/F_BACnet_EventTransitionFlags
FUNCTION F_BACnet_EventTransitionFlags : ST_BACnet_EventTransitionBits
VAR_INPUT
	data	: WORD;
END_VAR
VAR
END_VAR

F_BACnet_EventTransitionFlags.to_normal := _F_BACnet_IsBitFieldBitSet( data:=data, bitNbr:=BACnetEventTransitionBit_to_normal);
F_BACnet_EventTransitionFlags.to_offnormal := _F_BACnet_IsBitFieldBitSet( data:=data, bitNbr:=BACnetEventTransitionBit_to_offnormal);
F_BACnet_EventTransitionFlags.to_fault := _F_BACnet_IsBitFieldBitSet( data:=data, bitNbr:=BACnetEventTransitionBit_to_fault);

END_FUNCTION

// POUs/BACnet Helper/Flags/F_BACnet_GetEventTransFlagsData
FUNCTION F_BACnet_GetEventTransFlagsData : WORD
VAR_INPUT
	Flags	: ST_BACnet_EventTransitionBits;
END_VAR
VAR
END_VAR

F_BACnet_GetEventTransFlagsData := 16#0005;
IF Flags.to_normal THEN
	F_BACnet_GetEventTransFlagsData := DWORD_TO_WORD(_F_BACnet_SetBitFieldBit(ptrData:=ADR(F_BACnet_GetEventTransFlagsData), bitNbr:=BACnetEventTransitionBit_to_normal));
END_IF
IF Flags.to_offnormal THEN
	F_BACnet_GetEventTransFlagsData := DWORD_TO_WORD(_F_BACnet_SetBitFieldBit(ptrData:=ADR(F_BACnet_GetEventTransFlagsData), bitNbr:=BACnetEventTransitionBit_to_offnormal));
END_IF
IF Flags.to_fault THEN
	F_BACnet_GetEventTransFlagsData := DWORD_TO_WORD(_F_BACnet_SetBitFieldBit(ptrData:=ADR(F_BACnet_GetEventTransFlagsData), bitNbr:=BACnetEventTransitionBit_to_fault));
END_IF

END_FUNCTION

// POUs/BACnet Helper/Flags/F_BACnet_GetLimitEnFlagsData
FUNCTION F_BACnet_GetLimitEnFlagsData : WORD
VAR_INPUT
	Flags	: ST_BACnet_LimitEnable;
END_VAR
VAR
END_VAR

F_BACnet_GetLimitEnFlagsData := 16#0006;
IF Flags.highLimitEnable THEN
	F_BACnet_GetLimitEnFlagsData := DWORD_TO_WORD(_F_BACnet_SetBitFieldBit(ptrData:=ADR(F_BACnet_GetLimitEnFlagsData), bitNbr:=BACnetLimitEnableBits_highLimit));
END_IF
IF Flags.lowLimitEnable THEN
	F_BACnet_GetLimitEnFlagsData := DWORD_TO_WORD(_F_BACnet_SetBitFieldBit(ptrData:=ADR(F_BACnet_GetLimitEnFlagsData), bitNbr:=BACnetLimitEnableBits_lowLimit));
END_IF

END_FUNCTION

// POUs/BACnet Helper/Flags/F_BACnet_GetStatusFlagsData
FUNCTION F_BACnet_GetStatusFlagsData : WORD
VAR_INPUT
	Flags : ST_BACnet_StatusFlags;
END_VAR

F_BACnet_GetStatusFlagsData	:= 16#0004;
IF Flags.in_alarm THEN
	F_BACnet_GetStatusFlagsData := DWORD_TO_WORD(_F_BACnet_SetBitFieldBit(ptrData:=ADR(F_BACnet_GetStatusFlagsData), bitNbr:=BACnetStatusFlags_in_alarm));
END_IF
IF Flags.fault THEN
	F_BACnet_GetStatusFlagsData := DWORD_TO_WORD(_F_BACnet_SetBitFieldBit(ptrData:=ADR(F_BACnet_GetStatusFlagsData), bitNbr:=BACnetStatusFlags_fault));
END_IF
IF Flags.overridden THEN
	F_BACnet_GetStatusFlagsData := DWORD_TO_WORD(_F_BACnet_SetBitFieldBit(ptrData:=ADR(F_BACnet_GetStatusFlagsData), bitNbr:=BACnetStatusFlags_overridden));
END_IF
IF Flags.out_of_service THEN
	F_BACnet_GetStatusFlagsData := DWORD_TO_WORD(_F_BACnet_SetBitFieldBit(ptrData:=ADR(F_BACnet_GetStatusFlagsData), bitNbr:=BACnetStatusFlags_out_of_service));
END_IF

END_FUNCTION

// POUs/BACnet Helper/Flags/F_BACnet_LimitEnableFlags
FUNCTION F_BACnet_LimitEnableFlags : ST_BACnet_LimitEnable
VAR_INPUT
	data	: WORD;
END_VAR
VAR
END_VAR

F_BACnet_LimitEnableFlags.highLimitEnable := _F_BACnet_IsBitFieldBitSet( data:=data, bitNbr:=BACnetLimitEnableBits_highLimit);
F_BACnet_LimitEnableFlags.lowLimitEnable := _F_BACnet_IsBitFieldBitSet( data:=data, bitNbr:=BACnetLimitEnableBits_lowLimit);

END_FUNCTION

// POUs/BACnet Helper/Real/F_BACnet_RealEQ
FUNCTION F_BACnet_RealEQ : BOOL
VAR_INPUT
	fIn1	: REAL;
	fIn2	: REAL;
END_VAR
VAR
END_VAR

IF (F_BACnet_IsFinite(fIn1) <> F_BACnet_IsFinite(fIn2)) THEN
	F_BACnet_RealEQ := FALSE;
	RETURN;
END_IF
IF F_BACnet_IsFinite(fIn1) THEN
	IF (fIn1 <> fIn2) THEN
		F_BACnet_RealEQ := FALSE;
		RETURN;
	END_IF
END_IF
F_BACnet_RealEQ := TRUE;

END_FUNCTION

// POUs/BACnet Helper/Real/F_BACnet_RealGE
FUNCTION F_BACnet_RealGE : BOOL
VAR_INPUT
	fIn1	: REAL;
	fIn2	: REAL;
END_VAR
VAR
END_VAR

IF NOT (F_BACnet_IsFinite(fIn1) OR F_BACnet_IsFinite(fIn2)) THEN
	F_BACnet_RealGE := FALSE;
	RETURN;
END_IF
F_BACnet_RealGE := (fIn1 >= fIn2);

END_FUNCTION

// POUs/BACnet Helper/Real/F_BACnet_RealGT
FUNCTION F_BACnet_RealGT : BOOL
VAR_INPUT
	fIn1	: REAL;
	fIn2	: REAL;
END_VAR
VAR
END_VAR

IF NOT (F_BACnet_IsFinite(fIn1) OR F_BACnet_IsFinite(fIn2)) THEN
	F_BACnet_RealGT := FALSE;
	RETURN;
END_IF
F_BACnet_RealGT := (fIn1 > fIn2);

END_FUNCTION

// POUs/BACnet Helper/Real/F_BACnet_RealLE
FUNCTION F_BACnet_RealLE : BOOL
VAR_INPUT
	fIn1	: REAL;
	fIn2	: REAL;
END_VAR
VAR
END_VAR

IF NOT (F_BACnet_IsFinite(fIn1) OR F_BACnet_IsFinite(fIn2)) THEN
	F_BACnet_RealLE := FALSE;
	RETURN;
END_IF
F_BACnet_RealLE := (fIn1 <= fIn2);

END_FUNCTION

// POUs/BACnet Helper/Real/F_BACnet_RealLT
FUNCTION F_BACnet_RealLT : BOOL
VAR_INPUT
	fIn1	: REAL;
	fIn2	: REAL;
END_VAR
VAR
END_VAR

IF NOT (F_BACnet_IsFinite(fIn1) OR F_BACnet_IsFinite(fIn2)) THEN
	F_BACnet_RealLT := FALSE;
	RETURN;
END_IF
F_BACnet_RealLT := (fIn1 < fIn2);

END_FUNCTION

// POUs/BACnet Helper/Real/F_BACnet_RealNothing
FUNCTION F_BACnet_RealNothing : DWORD

F_BACnet_RealNothing:=16#7FFFFFFF;

END_FUNCTION

// POUs/BACnet Helper/Real/F_BACnet_RealPV
FUNCTION F_BACnet_RealPV : DWORD
VAR_INPUT
	bEnable	: BOOL; (* TRUE = commit to stack, FALSE = do-nothing *)
	bNull	: BOOL; (* TRUE = clear priority, FALSE = write value from input *)
	rValue	: REAL;
END_VAR
VAR
	pDword : POINTER TO DWORD;
END_VAR

IF (bEnable) THEN
	IF (bNull) THEN
		F_BACnet_RealPV := F_BACnet_RealNull();
	ELSE
		pDword := ADR(rValue);
		F_BACnet_RealPV := pDword^;
	END_IF
ELSE
	F_BACnet_RealPV := F_BACnet_RealNothing();
END_IF

END_FUNCTION

// POUs/BACnet Helper/Real/F_BACnet_RealToStr
FUNCTION F_BACnet_RealToStr : STRING
VAR_INPUT
	pValue	: POINTER TO REAL;
END_VAR
VAR
	fArg	: T_Arg;
	pDWORD	: POINTER TO DWORD;
END_VAR

fArg.cbLen := 4;
fArg.eType := ARGTYPE_REAL;
fArg.pData := pValue;
pDWORD := pValue;
IF IsFinite(fArg) THEN
	F_BACnet_RealToStr := REAL_TO_STRING(pValue^);
ELSE
	IF (pDWORD^ = 16#7FFF0000) THEN
		F_BACnet_RealToStr := '#NULL';
	ELSIF (pDWORD^ AND 16#80000000) = 16#80000000 THEN
		F_BACnet_RealToStr := '-#QNAN';
	ELSE
		F_BACnet_RealToStr := '#QNAN';
	END_IF
END_IF

END_FUNCTION

// POUs/BACnet Helper/F_BACnet_GetObjectListIndex
FUNCTION F_BACnet_GetObjectListIndex : DINT
VAR_INPUT
	tObjectId	: T_BACnet_ObjectIdentifier := 16#FFFFFFFF;
END_VAR

VAR
	iMax : DINT;
	i : DINT;
END_VAR
(*All VAR_IN_OUT variables have been moved to the end of the declaration due to compatibility reasons*)
VAR_IN_OUT
	stObjIDList	: ST_BACnet_ObjectIdentifierList;
END_VAR

iMax := UDINT_TO_DINT(stObjIDList.nEntries)-1;
F_BACnet_GetObjectListIndex := -1; (* preset: no match *)
FOR i := 0 TO iMax DO
	IF stObjIDList.arrObjList[i] = tObjectId THEN
		F_BACnet_GetObjectListIndex := i; (* match *)
		RETURN;
	END_IF
END_FOR

END_FUNCTION

// POUs/BACnet Logic/F_BinPV_AND
FUNCTION F_BinPV_AND : E_BACNETBINARYPV
VAR_INPUT
	eBinPV1:	E_BACNETBINARYPV;
	eBinPV2:	E_BACNETBINARYPV;
END_VAR
VAR
END_VAR

IF (eBinPV1 = eBinPV2) THEN
	F_BinPV_AND := eBinPV1;
ELSE
	F_BinPV_AND := BACnetBinaryPV_Nothing;
END_IF

END_FUNCTION

// POUs/BACnet Logic/F_BinPV_NOT
FUNCTION F_BinPV_NOT : E_BACNETBINARYPV
VAR_INPUT
	eBinPV:	E_BACNETBINARYPV;
END_VAR
VAR
END_VAR

IF (eBinPV = BACnetBinaryPV_active) THEN
	F_BinPV_NOT := BACnetBinaryPV_inactive;
ELSIF (eBinPV = BACnetBinaryPV_inactive) THEN
	F_BinPV_NOT := BACnetBinaryPV_active;
ELSE
	F_BinPV_NOT := eBinPV;
END_IF

END_FUNCTION

// POUs/BACnet Logic/F_BinPV_OR
FUNCTION F_BinPV_OR : E_BACNETBINARYPV
VAR_INPUT
	eBinPV1:	E_BACNETBINARYPV;
	eBinPV2:	E_BACNETBINARYPV;
END_VAR
VAR
END_VAR

IF (eBinPV1 = BACnetBinaryPV_active) OR (eBinPV2 = BACnetBinaryPV_active) THEN
	F_BinPV_OR := BACnetBinaryPV_active;
ELSIF (eBinPV1 = BACnetBinaryPV_inactive) OR (eBinPV2 = BACnetBinaryPV_inactive) THEN
	F_BinPV_OR := BACnetBinaryPV_inactive;
ELSIF (eBinPV1 = BACnetBinaryPV_NULL) OR (eBinPV2 = BACnetBinaryPV_NULL) THEN
	F_BinPV_OR := BACnetBinaryPV_NULL;
ELSE
	F_BinPV_OR := BACnetBinaryPV_Nothing;
END_IF

END_FUNCTION

// POUs/BACnet Logic/F_BinPV_To_Bool
FUNCTION F_BinPV_To_Bool : BOOL
VAR_INPUT
	eBinPV		: E_BACNETBINARYPV;
END_VAR
VAR
END_VAR

F_BinPV_To_Bool := (eBinPV = BACnetBinaryPV_active);

END_FUNCTION

// POUs/BACnet Logic/F_BinPV_XOR
FUNCTION F_BinPV_XOR : E_BACNETBINARYPV
VAR_INPUT
	eBinPV1:	E_BACNETBINARYPV;
	eBinPV2:	E_BACNETBINARYPV;
END_VAR
VAR
END_VAR

IF (eBinPV1 = BACnetBinaryPV_active) XOR (eBinPV2 = BACnetBinaryPV_active) THEN
	F_BinPV_XOR := BACnetBinaryPV_active;
ELSIF (eBinPV1 = BACnetBinaryPV_inactive) XOR (eBinPV2 = BACnetBinaryPV_inactive) THEN
	F_BinPV_XOR := BACnetBinaryPV_inactive;
ELSIF (eBinPV1 = BACnetBinaryPV_NULL) XOR (eBinPV2 = BACnetBinaryPV_NULL) THEN
	F_BinPV_XOR := BACnetBinaryPV_NULL;
ELSE
	F_BinPV_XOR := BACnetBinaryPV_Nothing;
END_IF

END_FUNCTION

// POUs/BACnet Logic/F_Bool_To_BinPV
FUNCTION F_Bool_To_BinPV : E_BACNETBINARYPV
VAR_INPUT
	bEnable	: BOOL;
	bNull	: BOOL;
	bBool	: BOOL;
END_VAR
VAR
END_VAR

IF (NOT bEnable) THEN
	F_Bool_To_BinPV := BACnetBinaryPV_Nothing;
ELSIF bNull THEN
	F_Bool_To_BinPV := BACnetBinaryPV_NULL;
ELSIF bBOOL THEN
	F_Bool_To_BinPV := BACnetBinaryPV_active;
ELSE
	F_Bool_To_BinPV := BACnetBinaryPV_inactive;
END_IF

END_FUNCTION

// POUs/BACnet Objects/Local (Server)/[Internal]/_FB_BACnet_AnalogObject
FUNCTION_BLOCK  _FB_BACnet_AnalogObject EXTENDS _FB_BACnet_Object
VAR_OUTPUT
	fPresentValue : REAL;
END_VAR

SUPER^(Device := Device);

END_FUNCTION_BLOCK

// POUs/BACnet Objects/Local (Server)/[Internal]/_FB_BACnet_Object
FUNCTION_BLOCK  _FB_BACnet_Object
VAR_IN_OUT
	Device			: FB_BACnet_Device;
END_VAR
VAR_OUTPUT
	bReady				: BOOL;
	bOverridden			: BOOL;
	bOutOfService		: BOOL;
	bFault				: BOOL;
	bInAlarm			: BOOL;
	bError				: BOOL;
	nErrorId			: UINT;
END_VAR
VAR
	_StatusFlags AT%I*:WORD;		(* ~(BACnet_StatusFlags		:		: )	*)
	_StatusFlagsBits : ST_BACnet_StatusFlags;
	_nUpdateCount : UDINT := 0;
END_VAR

(* update device *)
IF Device._nUpdateCount = _nUpdateCount THEN
	Device();
END_IF
(* remind current number of update counter *)
_nUpdateCount := Device._nUpdateCount;

IF _StatusFlags < 4 THEN
	(* mapping seems to be wrong (bit string for status flags must be 4 in minimum) *)
	nErrorId := BACnet_ERR_WRONG_MAPPING;

ELSIF Device.bOperational THEN
	(* clear error flag *)
	nErrorId := BACnet_ERR_NO_ERROR;
	bReady := TRUE;

	(* build bit states *)
	_StatusFlagsBits	:= F_BACnet_StatusFlags(_StatusFlags);

	(* copy states to output *)
	bOverridden := _StatusFlagsBits.overridden;
	bOutOfService := _StatusFlagsBits.out_of_service;
	bFault := _StatusFlagsBits.fault;
	bInAlarm := _StatusFlagsBits.in_alarm;
ELSE
	bReady := FALSE;
	(* and set error ID *)
	nErrorId := BACnet_ERR_OPERATIONAL;
END_IF

(* set error flag *)
bError := (nErrorId <> BACnet_ERR_NO_ERROR);

END_FUNCTION_BLOCK

// POUs/BACnet Objects/Local (Server)/[Internal]/_FB_BACnet_BinaryObject
FUNCTION_BLOCK  _FB_BACnet_BinaryObject EXTENDS _FB_BACnet_Object
VAR_OUTPUT
	bPresentValue	: BOOL;
END_VAR

SUPER^(Device := Device);

END_FUNCTION_BLOCK

// POUs/BACnet Objects/Local (Server)/ADS/FB_BACnet_AnalogOutput_ADS
FUNCTION_BLOCK FB_BACnet_AnalogOutput_ADS
VAR_INPUT
	bEnablePV			: BOOL; (* enable PV write commands *)
	bNullPV				: BOOL; (* clear priority entry *)
	fPV					: REAL; (* decimal number for priority x, when input bEnablePV is TRUE and bNullPV is FALSE *)
	bManual				: BOOL; (* FALSE --> TRUE: write present_value immediately, FALSE: only write present_value on-change, TRUE: write present_value on-change and when device turns operational *)
	ePriority			: E_BACNETPRIORITY := BACNETPRIORITY_12;
END_VAR
VAR_IN_OUT
	Device				: FB_BACnet_Device;
END_VAR
VAR_OUTPUT
	bReady				: BOOL;
	bPvDone				: BOOL; (* present_value written over ADS *)
	fPresentValue		: REAL;
	bOverridden			: BOOL;
	bOutOfService		: BOOL;
	bFault				: BOOL;
	bInAlarm			: BOOL;
	tObjectID			: T_BACnet_ObjectIdentifier := 16#FFFFFFFF;
	bError				: BOOL;
	nErrorId			: UINT;
	nAdsErrorId			: UDINT;
END_VAR
VAR
	_PresentValue AT%I*: REAL; 			(* ~(BACnet_PresentValue 		:		: )
								   			(BACnet_ObjectType 			: AO	: )	*)
    _PresentValue_Ads : DWORD;
	_ObjectId AT%I*: DWORD;				(* ~(BACnet_ObjectIdentifier	:		: LINK) *)
	_StatusFlags AT%I*: WORD; 			(* ~(BACnet_StatusFlags 		:		: )	*)
	_StatusFlagsBits : ST_BACnet_StatusFlags;
	_nUpdateCount : UDINT := 0;
	_WriteProp : FB_BACnet_WriteProp;
	_rtrigManual : R_TRIG;
	_bNullPvOld : BOOL;
	_nObjType : E_BACNETOBJECTTYPE;
END_VAR

(* update server device *)
IF (Device._nUpdateCount = _nUpdateCount) THEN
	Device();
END_IF
(* remind current number of update counter *)
_nUpdateCount := Device._nUpdateCount;

(* trigger on manual flag *)
_rtrigManual(CLK:= bManual, Q=> );

(* decode object type *)
_nObjType := F_BACnet_GetObjType(_ObjectId);

IF Device.bFirstCycle THEN
	(* first call of the server device since reboot/reset *)
	bReady := FALSE;
	bPvDone := FALSE;

ELSIF _nObjType <> BACnetObjectType_AnalogOutput THEN
	(* wrong mapped object type *)
	nErrorId := BACnet_ERR_INVALID_OBJECTTYPE;
	bReady := FALSE;
	bPvDone := FALSE;

ELSIF (_StatusFlags < 4) THEN
	(* wrong mapping *)
	nErrorId := BACnet_ERR_WRONG_MAPPING;
	bReady := FALSE;
	bPvDone := FALSE;

ELSIF Device.bOperational THEN

	IF Device.stAdsConn.bValid THEN
		(* write present_value on manual trigger, on-change and on operational recover *)
		IF		bEnablePV
			AND	(		_rtrigManual.Q
					OR	(MEMCMP(pBuf1:=ADR(fPV), pBuf2:=ADR(_PresentValue_Ads), n:=SIZEOF(_PresentValue_Ads)) <> 0)
					OR	((NOT bReady) AND bManual)
					OR	(bNullPV <> _bNullPvOld)
				)
		THEN
			_WriteProp.bExecute := TRUE;
			bPvDone := FALSE;
			(* write depending on enable state *)
			_PresentValue_Ads := F_BACnet_RealPV(TRUE, bNullPV, fPV);
			(* remind null flag *)
			_bNullPvOld := bNullPV;
		END_IF

		(* ready state *)
		IF (nAdsErrorId = 0) THEN
			bReady := TRUE;
			nErrorId := BACnet_ERR_NO_ERROR;
		END_IF

	ELSE
		(* invalid ADS connection *)
		bReady := FALSE;
		nErrorId := BACnet_ERR_INVALID_ADS_CONN;
		bPvDone := FALSE;
	END_IF

	(* present value *)
	fPresentValue := _PresentValue;

	(* build bit states *)
	_StatusFlagsBits := F_BACnet_StatusFlags(_StatusFlags);

	(* copy states to output *)
	bOverridden := _StatusFlagsBits.overridden;
	bOutOfService := _StatusFlagsBits.out_of_service;
	bFault := _StatusFlagsBits.fault;
	bInAlarm := _StatusFlagsBits.in_alarm;
	tObjectID := _ObjectId;

ELSE
	(* server device not ready, reset local ready also *)
	bReady := FALSE;
	nErrorId := BACnet_ERR_OPERATIONAL;
	bPvDone := FALSE;
END_IF

(* call write property command *)
_WriteProp(
	BACnetDevicePort	:= Device.stAdsConn.nAmsPort,
	bExecute			:= ,
	sNetId				:= Device.stAdsConn.sAmsNetId,
	ObjectType			:= _nObjType,
	PropertyID			:= BACnetPropertyIdentifier_PresentValue,
	Priority			:= ePriority,
	DataType			:= BACnetDataType_Real,
	ObjectInstance		:= F_BACnet_GetObjInstance(_ObjectId),
	ptrValue			:= ADR(_PresentValue_Ads),
	nLenValue			:= SIZEOF(_PresentValue_Ads),
	bDone				=> ,
	bBusy				=> ,
	bError				=> ,
	nErrID				=> );

(* set done flag *)
IF _WriteProp.bExecute AND (NOT _WriteProp.bBusy) THEN
	(* check if command was finished with error *)
	IF _WriteProp.bError THEN
		bPvDone		:= FALSE;
		bReady		:= FALSE;
		nErrorId	:= BACnet_ERR_ADS_Write;
	ELSE
		(* successful written *)
		bPvDone		:= TRUE;
	END_IF
	nAdsErrorId := _WriteProp.nErrID;
	(* reset execution bit *)
	_WriteProp(bExecute := FALSE);
END_IF

(* set error flag *)
bError := (nErrorId <> BACnet_ERR_NO_ERROR) OR (nAdsErrorId <> 0);

END_FUNCTION_BLOCK

// POUs/BACnet Objects/Local (Server)/ADS/FB_BACnet_AnalogValue_ADS
FUNCTION_BLOCK FB_BACnet_AnalogValue_ADS
VAR_INPUT
	bEnablePV			: BOOL; (* enable PV write commands *)
	bNullPV				: BOOL; (* clear priority entry *)
	fPV					: REAL; (* decimal number for priority x, when input bEnablePV is TRUE and bNullPV is FALSE *)
	bManual				: BOOL; (* FALSE --> TRUE: write present_value immediately, FALSE: only write present_value on-change, TRUE: write present_value on-change and when device turns operational *)
	ePriority			: E_BACNETPRIORITY := BACNETPRIORITY_12;
END_VAR
VAR_IN_OUT
	Device				: FB_BACnet_Device;
END_VAR
VAR_OUTPUT
	bReady				: BOOL;
	bPvDone				: BOOL; (* present_value written over ADS *)
	fPresentValue		: REAL;
	bOverridden			: BOOL;
	bOutOfService		: BOOL;
	bFault				: BOOL;
	bInAlarm			: BOOL;
	tObjectID			: T_BACnet_ObjectIdentifier := 16#FFFFFFFF;
	bError				: BOOL;
	nErrorId			: UINT;
	nAdsErrorId			: UDINT;
END_VAR
VAR
	_PresentValue AT%I*: REAL; 			(* ~(BACnet_PresentValue 		:		: )
								   			(BACnet_ObjectType 			: AV	: )	*)
	_ObjectId AT%I*: DWORD;				(* ~(BACnet_ObjectIdentifier	:		: LINK) *)
	_StatusFlags AT%I*: WORD; 			(* ~(BACnet_StatusFlags 		:		: )	*)
    _PresentValue_Ads : DWORD;
	_StatusFlagsBits : ST_BACnet_StatusFlags;
	_nUpdateCount : UDINT := 0;
	_WriteProp : FB_BACnet_WriteProp;
	_rtrigManual : R_TRIG;
	_bNullPvOld : BOOL;
	_nObjType : E_BACNETOBJECTTYPE;
END_VAR

(* update server device *)
IF (Device._nUpdateCount = _nUpdateCount) THEN
	Device();
END_IF
(* remind current number of update counter *)
_nUpdateCount := Device._nUpdateCount;

(* trigger on manual flag *)
_rtrigManual(CLK:= bManual, Q=> );

(* decode object type *)
_nObjType := F_BACnet_GetObjType(_ObjectId);

IF Device.bFirstCycle THEN
	(* first call of the server device since reboot/reset *)
	bReady := FALSE;
	bPvDone := FALSE;

ELSIF _nObjType <> BACnetObjectType_AnalogValue THEN
	(* wrong mapped object type *)
	nErrorId := BACnet_ERR_INVALID_OBJECTTYPE;
	bReady := FALSE;
	bPvDone := FALSE;

ELSIF (_StatusFlags < 4) THEN
	(* wrong mapping *)
	nErrorId := BACnet_ERR_WRONG_MAPPING;
	bReady := FALSE;
	bPvDone := FALSE;

ELSIF Device.bOperational THEN

	IF Device.stAdsConn.bValid THEN
		(* write present_value on manual trigger, on-change and on operational recover *)
		IF		bEnablePV
			AND	(		_rtrigManual.Q
					OR	(MEMCMP(pBuf1:=ADR(fPV), pBuf2:=ADR(_PresentValue_Ads), n:=SIZEOF(_PresentValue_Ads)) <> 0)
					OR	((NOT bReady) AND bManual)
					OR	(bNullPV <> _bNullPvOld)
				)
		THEN
			_WriteProp.bExecute := TRUE;
			bPvDone := FALSE;
			(* write depending on enable state *)
			_PresentValue_Ads := F_BACnet_RealPV(TRUE, bNullPV, fPV);
			(* remind null flag *)
			_bNullPvOld := bNullPV;
		END_IF

		(* ready state *)
		IF (nAdsErrorId = 0) THEN
			bReady := TRUE;
			nErrorId := BACnet_ERR_NO_ERROR;
		END_IF

	ELSE
		(* invalid ADS connection *)
		bReady := FALSE;
		nErrorId := BACnet_ERR_INVALID_ADS_CONN;
		bPvDone := FALSE;
	END_IF

	(* present value *)
	fPresentValue := _PresentValue;

	(* build bit states *)
	_StatusFlagsBits := F_BACnet_StatusFlags(_StatusFlags);

	(* copy states to output *)
	bOverridden := _StatusFlagsBits.overridden;
	bOutOfService := _StatusFlagsBits.out_of_service;
	bFault := _StatusFlagsBits.fault;
	bInAlarm := _StatusFlagsBits.in_alarm;
	tObjectID := _ObjectId;

ELSE
	(* server device not ready, reset local ready also *)
	bReady := FALSE;
	nErrorId := BACnet_ERR_OPERATIONAL;
	bPvDone := FALSE;
END_IF

(* call write property command *)
_WriteProp(
	BACnetDevicePort	:= Device.stAdsConn.nAmsPort,
	bExecute			:= ,
	sNetId				:= Device.stAdsConn.sAmsNetId,
	ObjectType			:= _nObjType,
	PropertyID			:= BACnetPropertyIdentifier_PresentValue,
	Priority			:= ePriority,
	DataType			:= BACnetDataType_Real,
	ObjectInstance		:= F_BACnet_GetObjInstance(_ObjectId),
	ptrValue			:= ADR(_PresentValue_Ads),
	nLenValue			:= SIZEOF(_PresentValue_Ads),
	bDone				=> ,
	bBusy				=> ,
	bError				=> ,
	nErrID				=> );

(* set done flag *)
IF _WriteProp.bExecute AND (NOT _WriteProp.bBusy) THEN
	(* check if command was finished with error *)
	IF _WriteProp.bError THEN
		bPvDone		:= FALSE;
		bReady		:= FALSE;
		nErrorId	:= BACnet_ERR_ADS_Write;
	ELSE
		(* successful written *)
		bPvDone		:= TRUE;
	END_IF
	nAdsErrorId := _WriteProp.nErrID;
	(* reset execution bit *)
	_WriteProp(bExecute := FALSE);
END_IF

(* set error flag *)
bError := (nErrorId <> BACnet_ERR_NO_ERROR) OR (nAdsErrorId <> 0);

END_FUNCTION_BLOCK

